	VAR jointtarget SDP_985 := [[-5.9, 34.76, 7.91, 0, 47.34, -89.94], [9E9, 9E9, 9E9, 9E9, 9E9, 9E9]];
	VAR jointtarget SDP_986 := [[-5.86, 34.75, 7.91, 0, 47.34, -91.23], [9E9, 9E9, 9E9, 9E9, 9E9, 9E9]];
	VAR jointtarget SDP_987 := [[-5.83, 34.75, 7.91, 0, 47.34, -92.52], [9E9, 9E9, 9E9, 9E9, 9E9, 9E9]];
	VAR jointtarget SDP_988 := [[-5.79, 34.75, 7.92, 0, 47.33, -93.81], [9E9, 9E9, 9E9, 9E9, 9E9, 9E9]];
	VAR jointtarget SDP_989 := [[-5.76, 34.75, 7.92, 0, 47.33, -95.1], [9E9, 9E9, 9E9, 9E9, 9E9, 9E9]];
	VAR jointtarget SDP_990 := [[-4.6, 34.64, 8.11, 0, 47.25, -94.6], [9E9, 9E9, 9E9, 9E9, 9E9, 9E9]];
	VAR jointtarget SDP_991 := [[-3.43, 34.55, 8.26, 0, 47.19, -93.43], [9E9, 9E9, 9E9, 9E9, 9E9, 9E9]];
	VAR jointtarget SDP_992 := [[-2.26, 34.49, 8.36, 0, 47.15, -92.26], [9E9, 9E9, 9E9, 9E9, 9E9, 9E9]];
	VAR jointtarget SDP_993 := [[-1.09, 34.45, 8.42, 0, 47.13, -91.09], [9E9, 9E9, 9E9, 9E9, 9E9, 9E9]];
	VAR jointtarget SDP_994 := [[0.09, 34.44, 8.44, 0, 47.12, -89.91], [9E9, 9E9, 9E9, 9E9, 9E9, 9E9]];
	VAR jointtarget SDP_995 := [[1.26, 34.46, 8.41, 0, 47.13, -88.74], [9E9, 9E9, 9E9, 9E9, 9E9, 9E9]];
	VAR jointtarget SDP_996 := [[2.43, 34.5, 8.35, 0, 47.16, -87.57], [9E9, 9E9, 9E9, 9E9, 9E9, 9E9]];
	VAR jointtarget SDP_997 := [[3.6, 34.56, 8.24, 0, 47.2, -86.4], [9E9, 9E9, 9E9, 9E9, 9E9, 9E9]];
	VAR jointtarget SDP_998 := [[4.77, 34.65, 8.08, 0, 47.27, -85.23], [9E9, 9E9, 9E9, 9E9, 9E9, 9E9]];
	VAR jointtarget SDP_999 := [[5.93, 34.77, 7.89, 0, 47.35, -84.07], [9E9, 9E9, 9E9, 9E9, 9E9, 9E9]];
	VAR jointtarget SDP_1000 := [[6.27, 34.83, 7.77, 0, 47.39, -79.23], [9E9, 9E9, 9E9, 9E9, 9E9, 9E9]];
	VAR jointtarget SDP_1001 := [[6.6, 34.96, 7.56, 0, 47.48, -69.9], [9E9, 9E9, 9E9, 9E9, 9E9, 9E9]];
	VAR jointtarget SDP_1002 := [[6.9, 35.14, 7.25, 0, 47.61, -60.6], [9E9, 9E9, 9E9, 9E9, 9E9, 9E9]];
	VAR jointtarget SDP_1003 := [[7.17, 35.37, 6.86, 0, 47.77, -51.33], [9E9, 9E9, 9E9, 9E9, 9E9, 9E9]];
	VAR jointtarget SDP_1004 := [[7.4, 35.64, 6.4, 0, 47.96, -42.1], [9E9, 9E9, 9E9, 9E9, 9E9, 9E9]];
	VAR jointtarget SDP_1005 := [[7.59, 35.95, 5.86, 0, 48.18, -32.91], [9E9, 9E9, 9E9, 9E9, 9E9, 9E9]];
	VAR jointtarget SDP_1006 := [[7.73, 36.29, 5.28, 0, 48.43, -23.77], [9E9, 9E9, 9E9, 9E9, 9E9, 9E9]];
	VAR jointtarget SDP_1007 := [[7.82, 36.65, 4.66, 0, 48.69, -14.68], [9E9, 9E9, 9E9, 9E9, 9E9, 9E9]];
	VAR jointtarget SDP_1008 := [[7.85, 37.02, 4.02, 0, 48.95, -5.65], [9E9, 9E9, 9E9, 9E9, 9E9, 9E9]];
	VAR jointtarget SDP_1009 := [[7.83, 37.4, 3.38, 0, 49.23, 3.33], [9E9, 9E9, 9E9, 9E9, 9E9, 9E9]];
	VAR jointtarget SDP_1010 := [[7.68, 38.65, 1.21, 0, 50.14, 7.68], [9E9, 9E9, 9E9, 9E9, 9E9, 9E9]];
	VAR jointtarget SDP_1011 := [[7.54, 39.92, -1.01, 0, 51.09, 7.54], [9E9, 9E9, 9E9, 9E9, 9E9, 9E9]];
	VAR jointtarget SDP_1012 := [[7.4, 41.21, -3.27, 0, 52.06, 7.4], [9E9, 9E9, 9E9, 9E9, 9E9, 9E9]];
	VAR jointtarget SDP_1013 := [[7.26, 42.52, -5.58, 0, 53.06, 7.26], [9E9, 9E9, 9E9, 9E9, 9E9, 9E9]];
	VAR jointtarget SDP_1014 := [[7.13, 43.85, -7.95, 0, 54.1, 7.13], [9E9, 9E9, 9E9, 9E9, 9E9, 9E9]];
	VAR jointtarget SDP_1015 := [[7.01, 45.21, -10.38, 0, 55.16, 7.01], [9E9, 9E9, 9E9, 9E9, 9E9, 9E9]];
	VAR jointtarget SDP_1016 := [[6.89, 46.6, -12.87, 0, 56.27, 6.89], [9E9, 9E9, 9E9, 9E9, 9E9, 9E9]];
	VAR jointtarget SDP_1017 := [[6.77, 48.03, -15.44, 0, 57.41, 6.77], [9E9, 9E9, 9E9, 9E9, 9E9, 9E9]];
	VAR jointtarget SDP_1018 := [[6.66, 49.49, -18.09, 0, 58.6, 6.66], [9E9, 9E9, 9E9, 9E9, 9E9, 9E9]];
	VAR jointtarget SDP_1019 := [[6.55, 51, -20.83, 0, 59.83, 6.55], [9E9, 9E9, 9E9, 9E9, 9E9, 9E9]];
	VAR jointtarget SDP_1020 := [[6.55, 51.04, -20.91, 0, 59.87, 5.89], [9E9, 9E9, 9E9, 9E9, 9E9, 9E9]];
	VAR jointtarget SDP_1021 := [[6.55, 51.09, -20.99, 0, 59.91, 4.56], [9E9, 9E9, 9E9, 9E9, 9E9, 9E9]];
	VAR jointtarget SDP_1022 := [[6.55, 51.13, -21.08, 0, 59.94, 3.24], [9E9, 9E9, 9E9, 9E9, 9E9, 9E9]];
	VAR jointtarget SDP_1023 := [[6.54, 51.18, -21.16, 0, 59.98, 1.91], [9E9, 9E9, 9E9, 9E9, 9E9, 9E9]];
	VAR jointtarget SDP_1024 := [[6.54, 51.22, -21.24, 0, 60.02, 0.59], [9E9, 9E9, 9E9, 9E9, 9E9, 9E9]];
	VAR jointtarget SDP_1025 := [[6.54, 51.27, -21.32, 0, 60.06, -0.74], [9E9, 9E9, 9E9, 9E9, 9E9, 9E9]];
	VAR jointtarget SDP_1026 := [[6.55, 51.32, -21.41, 0, 60.09, -2.06], [9E9, 9E9, 9E9, 9E9, 9E9, 9E9]];
	VAR jointtarget SDP_1027 := [[6.55, 51.36, -21.49, 0, 60.13, -3.38], [9E9, 9E9, 9E9, 9E9, 9E9, 9E9]];
	VAR jointtarget SDP_1028 := [[6.55, 51.41, -21.57, 0, 60.17, -4.7], [9E9, 9E9, 9E9, 9E9, 9E9, 9E9]];
	VAR jointtarget SDP_1029 := [[6.55, 51.45, -21.66, 0, 60.21, -6.03], [9E9, 9E9, 9E9, 9E9, 9E9, 9E9]];
	VAR jointtarget SDP_1030 := [[6.57, 51.63, -21.99, 0, 60.36, -6.68], [9E9, 9E9, 9E9, 9E9, 9E9, 9E9]];
	VAR jointtarget SDP_1031 := [[6.58, 51.82, -22.33, 0, 60.51, -6.66], [9E9, 9E9, 9E9, 9E9, 9E9, 9E9]];
	VAR jointtarget SDP_1032 := [[6.59, 52, -22.66, 0, 60.66, -6.65], [9E9, 9E9, 9E9, 9E9, 9E9, 9E9]];
	VAR jointtarget SDP_1033 := [[6.6, 52.19, -23, 0, 60.81, -6.64], [9E9, 9E9, 9E9, 9E9, 9E9, 9E9]];
	VAR jointtarget SDP_1034 := [[6.62, 52.37, -23.34, 0, 60.97, -6.62], [9E9, 9E9, 9E9, 9E9, 9E9, 9E9]];
	VAR jointtarget SDP_1035 := [[6.63, 52.56, -23.68, 0, 61.12, -6.61], [9E9, 9E9, 9E9, 9E9, 9E9, 9E9]];
	VAR jointtarget SDP_1036 := [[6.64, 52.75, -24.03, 0, 61.28, -6.6], [9E9, 9E9, 9E9, 9E9, 9E9, 9E9]];
	VAR jointtarget SDP_1037 := [[6.65, 52.94, -24.37, 0, 61.44, -6.59], [9E9, 9E9, 9E9, 9E9, 9E9, 9E9]];
	VAR jointtarget SDP_1038 := [[6.67, 53.13, -24.72, 0, 61.59, -6.57], [9E9, 9E9, 9E9, 9E9, 9E9, 9E9]];
	VAR jointtarget SDP_1039 := [[6.68, 53.32, -25.07, 0, 61.75, -6.56], [9E9, 9E9, 9E9, 9E9, 9E9, 9E9]];
	VAR jointtarget SDP_1040 := [[6.66, 53.69, -25.75, 0, 62.06, 3.75], [9E9, 9E9, 9E9, 9E9, 9E9, 9E9]];
	VAR jointtarget SDP_1041 := [[6.58, 54.03, -26.38, 0, 62.35, 24.31], [9E9, 9E9, 9E9, 9E9, 9E9, 9E9]];
	VAR jointtarget SDP_1042 := [[6.43, 54.3, -26.87, 0, 62.58, 44.81], [9E9, 9E9, 9E9, 9E9, 9E9, 9E9]];
	VAR jointtarget SDP_1043 := [[6.24, 54.46, -27.17, 0, 62.71, 65.27], [9E9, 9E9, 9E9, 9E9, 9E9, 9E9]];
	VAR jointtarget SDP_1044 := [[6.04, 54.49, -27.22, 0, 62.73, 85.71], [9E9, 9E9, 9E9, 9E9, 9E9, 9E9]];
	VAR jointtarget SDP_1045 := [[5.84, 54.38, -27.02, 0, 62.64, 106.16], [9E9, 9E9, 9E9, 9E9, 9E9, 9E9]];
	VAR jointtarget SDP_1046 := [[5.67, 54.15, -26.6, 0, 62.45, 126.64], [9E9, 9E9, 9E9, 9E9, 9E9, 9E9]];
	VAR jointtarget SDP_1047 := [[5.56, 53.83, -26.02, 0, 62.19, 147.18], [9E9, 9E9, 9E9, 9E9, 9E9, 9E9]];
	VAR jointtarget SDP_1048 := [[5.52, 53.47, -25.35, 0, 61.88, 167.78], [9E9, 9E9, 9E9, 9E9, 9E9, 9E9]];
	VAR jointtarget SDP_1049 := [[5.55, 53.1, -24.68, 0, 61.57, 188.46], [9E9, 9E9, 9E9, 9E9, 9E9, 9E9]];
	VAR jointtarget SDP_1050 := [[5.58, 52.92, -24.34, 0, 61.42, 198.82], [9E9, 9E9, 9E9, 9E9, 9E9, 9E9]];
	VAR jointtarget SDP_1051 := [[5.62, 52.74, -24.02, 0, 61.27, 198.86], [9E9, 9E9, 9E9, 9E9, 9E9, 9E9]];
	VAR jointtarget SDP_1052 := [[5.65, 52.56, -23.69, 0, 61.13, 198.89], [9E9, 9E9, 9E9, 9E9, 9E9, 9E9]];
	VAR jointtarget SDP_1053 := [[5.69, 52.39, -23.36, 0, 60.98, 198.93], [9E9, 9E9, 9E9, 9E9, 9E9, 9E9]];
	VAR jointtarget SDP_1054 := [[5.72, 52.21, -23.04, 0, 60.83, 198.96], [9E9, 9E9, 9E9, 9E9, 9E9, 9E9]];
	VAR jointtarget SDP_1055 := [[5.76, 52.03, -22.72, 0, 60.68, 199], [9E9, 9E9, 9E9, 9E9, 9E9, 9E9]];
	VAR jointtarget SDP_1056 := [[5.79, 51.86, -22.4, 0, 60.54, 199.03], [9E9, 9E9, 9E9, 9E9, 9E9, 9E9]];
	VAR jointtarget SDP_1057 := [[5.83, 51.68, -22.08, 0, 60.39, 199.07], [9E9, 9E9, 9E9, 9E9, 9E9, 9E9]];
	VAR jointtarget SDP_1058 := [[5.87, 51.51, -21.76, 0, 60.25, 199.11], [9E9, 9E9, 9E9, 9E9, 9E9, 9E9]];
	VAR jointtarget SDP_1059 := [[5.9, 51.33, -21.44, 0, 60.11, 199.14], [9E9, 9E9, 9E9, 9E9, 9E9, 9E9]];
	VAR jointtarget SDP_1060 := [[5.91, 51.29, -21.36, 0, 60.07, 198.49], [9E9, 9E9, 9E9, 9E9, 9E9, 9E9]];
	VAR jointtarget SDP_1061 := [[5.92, 51.25, -21.28, 0, 60.04, 197.17], [9E9, 9E9, 9E9, 9E9, 9E9, 9E9]];
	VAR jointtarget SDP_1062 := [[5.93, 51.2, -21.2, 0, 60, 195.86], [9E9, 9E9, 9E9, 9E9, 9E9, 9E9]];
	VAR jointtarget SDP_1063 := [[5.93, 51.16, -21.12, 0, 59.96, 194.54], [9E9, 9E9, 9E9, 9E9, 9E9, 9E9]];
	VAR jointtarget SDP_1064 := [[5.94, 51.11, -21.04, 0, 59.93, 193.22], [9E9, 9E9, 9E9, 9E9, 9E9, 9E9]];
	VAR jointtarget SDP_1065 := [[5.94, 51.07, -20.96, 0, 59.89, 191.9], [9E9, 9E9, 9E9, 9E9, 9E9, 9E9]];
	VAR jointtarget SDP_1066 := [[5.95, 51.03, -20.88, 0, 59.85, 190.58], [9E9, 9E9, 9E9, 9E9, 9E9, 9E9]];
	VAR jointtarget SDP_1067 := [[5.95, 50.98, -20.8, 0, 59.82, 189.26], [9E9, 9E9, 9E9, 9E9, 9E9, 9E9]];
	VAR jointtarget SDP_1068 := [[5.96, 50.94, -20.72, 0, 59.78, 187.94], [9E9, 9E9, 9E9, 9E9, 9E9, 9E9]];
	VAR jointtarget SDP_1069 := [[5.96, 50.89, -20.64, 0, 59.74, 186.62], [9E9, 9E9, 9E9, 9E9, 9E9, 9E9]];
	VAR jointtarget SDP_1070 := [[6.05, 49.48, -18.07, 0, 58.59, 186.05], [9E9, 9E9, 9E9, 9E9, 9E9, 9E9]];
	VAR jointtarget SDP_1071 := [[6.15, 48.11, -15.58, 0, 57.48, 186.15], [9E9, 9E9, 9E9, 9E9, 9E9, 9E9]];
	VAR jointtarget SDP_1072 := [[6.25, 46.77, -13.17, 0, 56.4, 186.25], [9E9, 9E9, 9E9, 9E9, 9E9, 9E9]];
	VAR jointtarget SDP_1073 := [[6.35, 45.46, -10.82, 0, 55.36, 186.35], [9E9, 9E9, 9E9, 9E9, 9E9, 9E9]];
	VAR jointtarget SDP_1074 := [[6.46, 44.18, -8.53, 0, 54.35, 186.46], [9E9, 9E9, 9E9, 9E9, 9E9, 9E9]];
	VAR jointtarget SDP_1075 := [[6.56, 42.92, -6.29, 0, 53.37, 186.56], [9E9, 9E9, 9E9, 9E9, 9E9, 9E9]];
	VAR jointtarget SDP_1076 := [[6.68, 41.68, -4.11, 0, 52.43, 186.68], [9E9, 9E9, 9E9, 9E9, 9E9, 9E9]];
	VAR jointtarget SDP_1077 := [[6.79, 40.47, -1.97, 0, 51.5, 186.79], [9E9, 9E9, 9E9, 9E9, 9E9, 9E9]];
	VAR jointtarget SDP_1078 := [[6.91, 39.27, 0.13, 0, 50.6, 186.91], [9E9, 9E9, 9E9, 9E9, 9E9, 9E9]];
	VAR jointtarget SDP_1079 := [[7.04, 38.08, 2.19, 0, 49.73, 187.04], [9E9, 9E9, 9E9, 9E9, 9E9, 9E9]];
	VAR jointtarget SDP_1080 := [[7.05, 37.71, 2.84, 0, 49.45, 182.55], [9E9, 9E9, 9E9, 9E9, 9E9, 9E9]];
	VAR jointtarget SDP_1081 := [[7.02, 37.33, 3.48, 0, 49.18, 173.52], [9E9, 9E9, 9E9, 9E9, 9E9, 9E9]];
	VAR jointtarget SDP_1082 := [[6.93, 36.97, 4.11, 0, 48.92, 164.43], [9E9, 9E9, 9E9, 9E9, 9E9, 9E9]];
	VAR jointtarget SDP_1083 := [[6.78, 36.63, 4.69, 0, 48.68, 155.28], [9E9, 9E9, 9E9, 9E9, 9E9, 9E9]];
	VAR jointtarget SDP_1084 := [[6.6, 36.33, 5.22, 0, 48.45, 146.1], [9E9, 9E9, 9E9, 9E9, 9E9, 9E9]];
	VAR jointtarget SDP_1085 := [[6.36, 36.05, 5.69, 0, 48.26, 136.86], [9E9, 9E9, 9E9, 9E9, 9E9, 9E9]];
	VAR jointtarget SDP_1086 := [[6.09, 35.83, 6.08, 0, 48.1, 127.59], [9E9, 9E9, 9E9, 9E9, 9E9, 9E9]];
	VAR jointtarget SDP_1087 := [[5.79, 35.65, 6.38, 0, 47.97, 118.29], [9E9, 9E9, 9E9, 9E9, 9E9, 9E9]];
	VAR jointtarget SDP_1088 := [[5.47, 35.53, 6.58, 0, 47.89, 108.97], [9E9, 9E9, 9E9, 9E9, 9E9, 9E9]];
	VAR jointtarget SDP_1089 := [[5.13, 35.47, 6.69, 0, 47.84, 99.63], [9E9, 9E9, 9E9, 9E9, 9E9, 9E9]];
	VAR jointtarget SDP_1090 := [[4.07, 35.38, 6.85, 0, 47.78, 94.07], [9E9, 9E9, 9E9, 9E9, 9E9, 9E9]];
	VAR jointtarget SDP_1091 := [[3.01, 35.31, 6.97, 0, 47.73, 93.01], [9E9, 9E9, 9E9, 9E9, 9E9, 9E9]];
	VAR jointtarget SDP_1092 := [[1.95, 35.26, 7.05, 0, 47.69, 91.95], [9E9, 9E9, 9E9, 9E9, 9E9, 9E9]];
	VAR jointtarget SDP_1093 := [[0.89, 35.23, 7.1, 0, 47.67, 90.89], [9E9, 9E9, 9E9, 9E9, 9E9, 9E9]];
	VAR jointtarget SDP_1094 := [[-0.18, 35.22, 7.11, 0, 47.67, 89.82], [9E9, 9E9, 9E9, 9E9, 9E9, 9E9]];
	VAR jointtarget SDP_1095 := [[-1.24, 35.24, 7.09, 0, 47.68, 88.76], [9E9, 9E9, 9E9, 9E9, 9E9, 9E9]];
	VAR jointtarget SDP_1096 := [[-2.31, 35.27, 7.03, 0, 47.7, 87.69], [9E9, 9E9, 9E9, 9E9, 9E9, 9E9]];
	VAR jointtarget SDP_1097 := [[-3.37, 35.33, 6.93, 0, 47.74, 86.63], [9E9, 9E9, 9E9, 9E9, 9E9, 9E9]];
	VAR jointtarget SDP_1098 := [[-4.43, 35.41, 6.8, 0, 47.8, 85.57], [9E9, 9E9, 9E9, 9E9, 9E9, 9E9]];
	VAR jointtarget SDP_1099 := [[-5.48, 35.5, 6.63, 0, 47.87, 84.52], [9E9, 9E9, 9E9, 9E9, 9E9, 9E9]];
	VAR jointtarget SDP_1100 := [[-5.59, 35.51, 6.62, 0, 47.87, 86.6], [9E9, 9E9, 9E9, 9E9, 9E9, 9E9]];
	VAR jointtarget SDP_1101 := [[-5.71, 35.51, 6.62, 0, 47.87, 90.88], [9E9, 9E9, 9E9, 9E9, 9E9, 9E9]];
	VAR jointtarget SDP_1102 := [[-5.82, 35.5, 6.64, 0, 47.86, 95.15], [9E9, 9E9, 9E9, 9E9, 9E9, 9E9]];
	VAR jointtarget SDP_1103 := [[-5.93, 35.48, 6.67, 0, 47.85, 99.43], [9E9, 9E9, 9E9, 9E9, 9E9, 9E9]];
	VAR jointtarget SDP_1104 := [[-6.04, 35.45, 6.72, 0, 47.83, 103.71], [9E9, 9E9, 9E9, 9E9, 9E9, 9E9]];
	VAR jointtarget SDP_1105 := [[-6.14, 35.41, 6.79, 0, 47.8, 107.99], [9E9, 9E9, 9E9, 9E9, 9E9, 9E9]];
	VAR jointtarget SDP_1106 := [[-6.25, 35.37, 6.86, 0, 47.77, 112.27], [9E9, 9E9, 9E9, 9E9, 9E9, 9E9]];
	VAR jointtarget SDP_1107 := [[-6.35, 35.31, 6.96, 0, 47.73, 116.56], [9E9, 9E9, 9E9, 9E9, 9E9, 9E9]];
	VAR jointtarget SDP_1108 := [[-6.44, 35.25, 7.06, 0, 47.69, 120.85], [9E9, 9E9, 9E9, 9E9, 9E9, 9E9]];
	VAR jointtarget SDP_1109 := [[-6.54, 35.18, 7.18, 0, 47.64, 125.15], [9E9, 9E9, 9E9, 9E9, 9E9, 9E9]];
	VAR jointtarget SDP_1110 := [[-6.59, 35.14, 7.25, 0, 47.61, 127.29], [9E9, 9E9, 9E9, 9E9, 9E9, 9E9]];
	VAR jointtarget SDP_1111 := [[-6.64, 35.09, 7.33, 0, 47.58, 127.23], [9E9, 9E9, 9E9, 9E9, 9E9, 9E9]];
	VAR jointtarget SDP_1112 := [[-6.7, 35.05, 7.4, 0, 47.55, 127.18], [9E9, 9E9, 9E9, 9E9, 9E9, 9E9]];
	VAR jointtarget SDP_1113 := [[-6.75, 35.01, 7.48, 0, 47.52, 127.12], [9E9, 9E9, 9E9, 9E9, 9E9, 9E9]];
	VAR jointtarget SDP_1114 := [[-6.81, 34.96, 7.55, 0, 47.48, 127.07], [9E9, 9E9, 9E9, 9E9, 9E9, 9E9]];
	VAR jointtarget SDP_1115 := [[-6.86, 34.92, 7.63, 0, 47.45, 127.01], [9E9, 9E9, 9E9, 9E9, 9E9, 9E9]];
	VAR jointtarget SDP_1116 := [[-6.92, 34.88, 7.7, 0, 47.42, 126.96], [9E9, 9E9, 9E9, 9E9, 9E9, 9E9]];
	VAR jointtarget SDP_1117 := [[-6.97, 34.83, 7.77, 0, 47.39, 126.91], [9E9, 9E9, 9E9, 9E9, 9E9, 9E9]];
	VAR jointtarget SDP_1118 := [[-7.03, 34.79, 7.85, 0, 47.36, 126.85], [9E9, 9E9, 9E9, 9E9, 9E9, 9E9]];
	VAR jointtarget SDP_1119 := [[-7.08, 34.75, 7.92, 0, 47.33, 126.8], [9E9, 9E9, 9E9, 9E9, 9E9, 9E9]];
	VAR jointtarget SDP_1120 := [[-7.39, 34.61, 8.16, 0, 47.24, 113.1], [9E9, 9E9, 9E9, 9E9, 9E9, 9E9]];
	VAR jointtarget SDP_1121 := [[-7.72, 34.63, 8.12, 0, 47.25, 85.99], [9E9, 9E9, 9E9, 9E9, 9E9, 9E9]];
	VAR jointtarget SDP_1122 := [[-8.01, 34.81, 7.81, 0, 47.38, 58.93], [9E9, 9E9, 9E9, 9E9, 9E9, 9E9]];
	VAR jointtarget SDP_1123 := [[-8.18, 35.11, 7.3, 0, 47.59, 31.98], [9E9, 9E9, 9E9, 9E9, 9E9, 9E9]];
	VAR jointtarget SDP_1124 := [[-8.21, 35.46, 6.71, 0, 47.84, 5.18], [9E9, 9E9, 9E9, 9E9, 9E9, 9E9]];
	VAR jointtarget SDP_1125 := [[-8.09, 35.79, 6.14, 0, 48.07, -21.48], [9E9, 9E9, 9E9, 9E9, 9E9, 9E9]];
	VAR jointtarget SDP_1126 := [[-7.85, 36.02, 5.74, 0, 48.24, -48.01], [9E9, 9E9, 9E9, 9E9, 9E9, 9E9]];
	VAR jointtarget SDP_1127 := [[-7.53, 36.12, 5.58, 0, 48.3, -74.47], [9E9, 9E9, 9E9, 9E9, 9E9, 9E9]];
	VAR jointtarget SDP_1128 := [[-7.21, 36.05, 5.7, 0, 48.26, -100.93], [9E9, 9E9, 9E9, 9E9, 9E9, 9E9]];
	VAR jointtarget SDP_1129 := [[-6.96, 35.83, 6.06, 0, 48.1, -127.44], [9E9, 9E9, 9E9, 9E9, 9E9, 9E9]];
	VAR jointtarget SDP_1130 := [[-6.9, 35.76, 6.19, 0, 48.05, -140.78], [9E9, 9E9, 9E9, 9E9, 9E9, 9E9]];
	VAR jointtarget SDP_1131 := [[-6.85, 35.69, 6.31, 0, 48, -140.72], [9E9, 9E9, 9E9, 9E9, 9E9, 9E9]];
	VAR jointtarget SDP_1132 := [[-6.79, 35.62, 6.43, 0, 47.95, -140.67], [9E9, 9E9, 9E9, 9E9, 9E9, 9E9]];
	VAR jointtarget SDP_1133 := [[-6.74, 35.55, 6.55, 0, 47.9, -140.62], [9E9, 9E9, 9E9, 9E9, 9E9, 9E9]];
	VAR jointtarget SDP_1134 := [[-6.68, 35.48, 6.67, 0, 47.85, -140.56], [9E9, 9E9, 9E9, 9E9, 9E9, 9E9]];
	VAR jointtarget SDP_1135 := [[-6.63, 35.41, 6.8, 0, 47.8, -140.51], [9E9, 9E9, 9E9, 9E9, 9E9, 9E9]];
	VAR jointtarget SDP_1136 := [[-6.58, 35.34, 6.92, 0, 47.75, -140.45], [9E9, 9E9, 9E9, 9E9, 9E9, 9E9]];
	VAR jointtarget SDP_1137 := [[-6.52, 35.26, 7.04, 0, 47.7, -140.4], [9E9, 9E9, 9E9, 9E9, 9E9, 9E9]];
	VAR jointtarget SDP_1138 := [[-6.47, 35.19, 7.16, 0, 47.65, -140.34], [9E9, 9E9, 9E9, 9E9, 9E9, 9E9]];
	VAR jointtarget SDP_1139 := [[-6.41, 35.12, 7.28, 0, 47.6, -140.29], [9E9, 9E9, 9E9, 9E9, 9E9, 9E9]];
	VAR jointtarget SDP_1140 := [[-6.38, 35.09, 7.33, 0, 47.58, -139.16], [9E9, 9E9, 9E9, 9E9, 9E9, 9E9]];
	VAR jointtarget SDP_1141 := [[-6.36, 35.06, 7.38, 0, 47.55, -136.92], [9E9, 9E9, 9E9, 9E9, 9E9, 9E9]];
	VAR jointtarget SDP_1142 := [[-6.33, 35.03, 7.43, 0, 47.53, -134.69], [9E9, 9E9, 9E9, 9E9, 9E9, 9E9]];
	VAR jointtarget SDP_1143 := [[-6.3, 35, 7.48, 0, 47.51, -132.45], [9E9, 9E9, 9E9, 9E9, 9E9, 9E9]];
	VAR jointtarget SDP_1144 := [[-6.27, 34.98, 7.53, 0, 47.5, -130.22], [9E9, 9E9, 9E9, 9E9, 9E9, 9E9]];
	VAR jointtarget SDP_1145 := [[-6.24, 34.95, 7.57, 0, 47.48, -127.98], [9E9, 9E9, 9E9, 9E9, 9E9, 9E9]];
	VAR jointtarget SDP_1146 := [[-6.21, 34.92, 7.61, 0, 47.46, -125.74], [9E9, 9E9, 9E9, 9E9, 9E9, 9E9]];
	VAR jointtarget SDP_1147 := [[-6.18, 34.9, 7.65, 0, 47.45, -123.5], [9E9, 9E9, 9E9, 9E9, 9E9, 9E9]];
	VAR jointtarget SDP_1148 := [[-6.14, 34.88, 7.69, 0, 47.43, -121.26], [9E9, 9E9, 9E9, 9E9, 9E9, 9E9]];
	VAR jointtarget SDP_1149 := [[-6.11, 34.86, 7.72, 0, 47.42, -119.01], [9E9, 9E9, 9E9, 9E9, 9E9, 9E9]];
	VAR jointtarget SDP_1150 := [[-6.09, 34.85, 7.74, 0, 47.42, -117.89], [9E9, 9E9, 9E9, 9E9, 9E9, 9E9]];
	VAR jointtarget SDP_1151 := [[-6.07, 34.84, 7.75, 0, 47.41, -117.87], [9E9, 9E9, 9E9, 9E9, 9E9, 9E9]];
	VAR jointtarget SDP_1152 := [[-6.05, 34.83, 7.77, 0, 47.4, -117.86], [9E9, 9E9, 9E9, 9E9, 9E9, 9E9]];
	VAR jointtarget SDP_1153 := [[-6.04, 34.81, 7.79, 0, 47.4, -117.84], [9E9, 9E9, 9E9, 9E9, 9E9, 9E9]];
	VAR jointtarget SDP_1154 := [[-6.02, 34.8, 7.8, 0, 47.39, -117.82], [9E9, 9E9, 9E9, 9E9, 9E9, 9E9]];
	VAR jointtarget SDP_1155 := [[-6, 34.79, 7.82, 0, 47.39, -117.8], [9E9, 9E9, 9E9, 9E9, 9E9, 9E9]];
	VAR jointtarget SDP_1156 := [[-5.98, 34.78, 7.84, 0, 47.38, -117.79], [9E9, 9E9, 9E9, 9E9, 9E9, 9E9]];
	VAR jointtarget SDP_1157 := [[-5.97, 34.77, 7.85, 0, 47.37, -117.77], [9E9, 9E9, 9E9, 9E9, 9E9, 9E9]];
	VAR jointtarget SDP_1158 := [[-5.95, 34.76, 7.87, 0, 47.37, -117.75], [9E9, 9E9, 9E9, 9E9, 9E9, 9E9]];
	VAR jointtarget SDP_1159 := [[-5.93, 34.75, 7.89, 0, 47.36, -117.73], [9E9, 9E9, 9E9, 9E9, 9E9, 9E9]];
	VAR jointtarget SDP_1160 := [[-4.75, 34.64, 8.08, 0, 47.28, -94.75], [9E9, 9E9, 9E9, 9E9, 9E9, 9E9]];
	VAR jointtarget SDP_1161 := [[-3.57, 34.55, 8.24, 0, 47.22, -93.57], [9E9, 9E9, 9E9, 9E9, 9E9, 9E9]];
	VAR jointtarget SDP_1162 := [[-2.38, 34.48, 8.35, 0, 47.17, -92.38], [9E9, 9E9, 9E9, 9E9, 9E9, 9E9]];
	VAR jointtarget SDP_1163 := [[-1.19, 34.44, 8.41, 0, 47.14, -91.19], [9E9, 9E9, 9E9, 9E9, 9E9, 9E9]];
	VAR jointtarget SDP_1164 := [[0, 34.43, 8.44, 0, 47.14, -90], [9E9, 9E9, 9E9, 9E9, 9E9, 9E9]];
	VAR jointtarget SDP_1165 := [[1.19, 34.44, 8.41, 0, 47.14, -88.81], [9E9, 9E9, 9E9, 9E9, 9E9, 9E9]];
	VAR jointtarget SDP_1166 := [[2.38, 34.48, 8.35, 0, 47.17, -87.62], [9E9, 9E9, 9E9, 9E9, 9E9, 9E9]];
	VAR jointtarget SDP_1167 := [[3.57, 34.55, 8.24, 0, 47.22, -86.43], [9E9, 9E9, 9E9, 9E9, 9E9, 9E9]];
	VAR jointtarget SDP_1168 := [[4.75, 34.64, 8.08, 0, 47.28, -85.25], [9E9, 9E9, 9E9, 9E9, 9E9, 9E9]];
	VAR jointtarget SDP_1169 := [[5.93, 34.75, 7.89, 0, 47.36, -84.07], [9E9, 9E9, 9E9, 9E9, 9E9, 9E9]];
	VAR jointtarget SDP_1170 := [[6.27, 34.82, 7.77, 0, 47.41, -79.23], [9E9, 9E9, 9E9, 9E9, 9E9, 9E9]];
	VAR jointtarget SDP_1171 := [[6.6, 34.94, 7.56, 0, 47.5, -69.9], [9E9, 9E9, 9E9, 9E9, 9E9, 9E9]];
	VAR jointtarget SDP_1172 := [[6.9, 35.12, 7.25, 0, 47.62, -60.6], [9E9, 9E9, 9E9, 9E9, 9E9, 9E9]];
	VAR jointtarget SDP_1173 := [[7.17, 35.35, 6.86, 0, 47.79, -51.33], [9E9, 9E9, 9E9, 9E9, 9E9, 9E9]];
	VAR jointtarget SDP_1174 := [[7.4, 35.63, 6.39, 0, 47.98, -42.1], [9E9, 9E9, 9E9, 9E9, 9E9, 9E9]];
	VAR jointtarget SDP_1175 := [[7.59, 35.94, 5.86, 0, 48.2, -32.91], [9E9, 9E9, 9E9, 9E9, 9E9, 9E9]];
	VAR jointtarget SDP_1176 := [[7.73, 36.28, 5.28, 0, 48.44, -23.77], [9E9, 9E9, 9E9, 9E9, 9E9, 9E9]];
	VAR jointtarget SDP_1177 := [[7.82, 36.64, 4.66, 0, 48.7, -14.68], [9E9, 9E9, 9E9, 9E9, 9E9, 9E9]];
	VAR jointtarget SDP_1178 := [[7.85, 37.01, 4.02, 0, 48.97, -5.65], [9E9, 9E9, 9E9, 9E9, 9E9, 9E9]];
	VAR jointtarget SDP_1179 := [[7.83, 37.38, 3.38, 0, 49.24, 3.33], [9E9, 9E9, 9E9, 9E9, 9E9, 9E9]];
	VAR jointtarget SDP_1180 := [[7.68, 38.61, 1.24, 0, 50.14, 7.68], [9E9, 9E9, 9E9, 9E9, 9E9, 9E9]];
	VAR jointtarget SDP_1181 := [[7.54, 39.86, -0.93, 0, 51.07, 7.54], [9E9, 9E9, 9E9, 9E9, 9E9, 9E9]];
	VAR jointtarget SDP_1182 := [[7.4, 41.12, -3.15, 0, 52.02, 7.4], [9E9, 9E9, 9E9, 9E9, 9E9, 9E9]];
	VAR jointtarget SDP_1183 := [[7.27, 42.41, -5.42, 0, 53.01, 7.27], [9E9, 9E9, 9E9, 9E9, 9E9, 9E9]];
	VAR jointtarget SDP_1184 := [[7.15, 43.72, -7.74, 0, 54.02, 7.15], [9E9, 9E9, 9E9, 9E9, 9E9, 9E9]];
	VAR jointtarget SDP_1185 := [[7.02, 45.05, -10.12, 0, 55.06, 7.02], [9E9, 9E9, 9E9, 9E9, 9E9, 9E9]];
	VAR jointtarget SDP_1186 := [[6.9, 46.42, -12.56, 0, 56.14, 6.9], [9E9, 9E9, 9E9, 9E9, 9E9, 9E9]];
	VAR jointtarget SDP_1187 := [[6.79, 47.81, -15.07, 0, 57.26, 6.79], [9E9, 9E9, 9E9, 9E9, 9E9, 9E9]];
	VAR jointtarget SDP_1188 := [[6.68, 49.24, -17.66, 0, 58.42, 6.68], [9E9, 9E9, 9E9, 9E9, 9E9, 9E9]];
	VAR jointtarget SDP_1189 := [[6.57, 50.72, -20.34, 0, 59.62, 6.57], [9E9, 9E9, 9E9, 9E9, 9E9, 9E9]];
	VAR jointtarget SDP_1190 := [[6.56, 50.86, -20.6, 0, 59.74, 8.75], [9E9, 9E9, 9E9, 9E9, 9E9, 9E9]];
	VAR jointtarget SDP_1191 := [[6.54, 51.01, -20.87, 0, 59.86, 13.12], [9E9, 9E9, 9E9, 9E9, 9E9, 9E9]];
	VAR jointtarget SDP_1192 := [[6.51, 51.15, -21.13, 0, 59.98, 17.48], [9E9, 9E9, 9E9, 9E9, 9E9, 9E9]];
	VAR jointtarget SDP_1193 := [[6.48, 51.29, -21.39, 0, 60.09, 21.83], [9E9, 9E9, 9E9, 9E9, 9E9, 9E9]];
	VAR jointtarget SDP_1194 := [[6.44, 51.43, -21.63, 0, 60.21, 26.18], [9E9, 9E9, 9E9, 9E9, 9E9, 9E9]];
	VAR jointtarget SDP_1195 := [[6.39, 51.56, -21.87, 0, 60.31, 30.52], [9E9, 9E9, 9E9, 9E9, 9E9, 9E9]];
	VAR jointtarget SDP_1196 := [[6.34, 51.68, -22.1, 0, 60.42, 34.86], [9E9, 9E9, 9E9, 9E9, 9E9, 9E9]];
	VAR jointtarget SDP_1197 := [[6.28, 51.8, -22.31, 0, 60.51, 39.19], [9E9, 9E9, 9E9, 9E9, 9E9, 9E9]];
	VAR jointtarget SDP_1198 := [[6.22, 51.91, -22.51, 0, 60.61, 43.51], [9E9, 9E9, 9E9, 9E9, 9E9, 9E9]];
	VAR jointtarget SDP_1199 := [[6.15, 52.01, -22.7, 0, 60.69, 47.83], [9E9, 9E9, 9E9, 9E9, 9E9, 9E9]];
	VAR jointtarget SDP_1200 := [[6.11, 52.07, -22.81, 0, 60.74, 49.99], [9E9, 9E9, 9E9, 9E9, 9E9, 9E9]];
	VAR jointtarget SDP_1201 := [[6.07, 52.13, -22.92, 0, 60.79, 49.95], [9E9, 9E9, 9E9, 9E9, 9E9, 9E9]];
	VAR jointtarget SDP_1202 := [[6.03, 52.19, -23.03, 0, 60.84, 49.9], [9E9, 9E9, 9E9, 9E9, 9E9, 9E9]];
	VAR jointtarget SDP_1203 := [[5.99, 52.25, -23.14, 0, 60.89, 49.86], [9E9, 9E9, 9E9, 9E9, 9E9, 9E9]];
	VAR jointtarget SDP_1204 := [[5.94, 52.31, -23.25, 0, 60.94, 49.82], [9E9, 9E9, 9E9, 9E9, 9E9, 9E9]];
	VAR jointtarget SDP_1205 := [[5.9, 52.37, -23.36, 0, 60.99, 49.78], [9E9, 9E9, 9E9, 9E9, 9E9, 9E9]];
	VAR jointtarget SDP_1206 := [[5.86, 52.43, -23.47, 0, 61.04, 49.74], [9E9, 9E9, 9E9, 9E9, 9E9, 9E9]];
	VAR jointtarget SDP_1207 := [[5.82, 52.49, -23.58, 0, 61.09, 49.7], [9E9, 9E9, 9E9, 9E9, 9E9, 9E9]];
	VAR jointtarget SDP_1208 := [[5.78, 52.55, -23.69, 0, 61.14, 49.66], [9E9, 9E9, 9E9, 9E9, 9E9, 9E9]];
	VAR jointtarget SDP_1209 := [[5.74, 52.61, -23.8, 0, 61.19, 49.61], [9E9, 9E9, 9E9, 9E9, 9E9, 9E9]];
	VAR jointtarget SDP_1210 := [[5.58, 52.98, -24.48, 0, 61.5, 36.07], [9E9, 9E9, 9E9, 9E9, 9E9, 9E9]];
	VAR jointtarget SDP_1211 := [[5.54, 53.44, -25.31, 0, 61.88, 9.25], [9E9, 9E9, 9E9, 9E9, 9E9, 9E9]];
	VAR jointtarget SDP_1212 := [[5.62, 53.88, -26.13, 0, 62.25, -17.44], [9E9, 9E9, 9E9, 9E9, 9E9, 9E9]];
	VAR jointtarget SDP_1213 := [[5.8, 54.22, -26.75, 0, 62.53, -44.04], [9E9, 9E9, 9E9, 9E9, 9E9, 9E9]];
	VAR jointtarget SDP_1214 := [[6.04, 54.38, -27.04, 0, 62.66, -70.57], [9E9, 9E9, 9E9, 9E9, 9E9, 9E9]];
	VAR jointtarget SDP_1215 := [[6.3, 54.32, -26.93, 0, 62.61, -97.09], [9E9, 9E9, 9E9, 9E9, 9E9, 9E9]];
	VAR jointtarget SDP_1216 := [[6.51, 54.06, -26.45, 0, 62.39, -123.65], [9E9, 9E9, 9E9, 9E9, 9E9, 9E9]];
	VAR jointtarget SDP_1217 := [[6.64, 53.65, -25.7, 0, 62.05, -150.3], [9E9, 9E9, 9E9, 9E9, 9E9, 9E9]];
	VAR jointtarget SDP_1218 := [[6.66, 53.18, -24.85, 0, 61.66, -177.06], [9E9, 9E9, 9E9, 9E9, 9E9, 9E9]];
	VAR jointtarget SDP_1219 := [[6.55, 52.76, -24.08, 0, 61.31, -203.94], [9E9, 9E9, 9E9, 9E9, 9E9, 9E9]];
	VAR jointtarget SDP_1220 := [[6.52, 52.69, -23.94, 0, 61.25, -217.36], [9E9, 9E9, 9E9, 9E9, 9E9, 9E9]];
	VAR jointtarget SDP_1221 := [[6.48, 52.62, -23.81, 0, 61.19, -217.39], [9E9, 9E9, 9E9, 9E9, 9E9, 9E9]];
	VAR jointtarget SDP_1222 := [[6.45, 52.54, -23.67, 0, 61.13, -217.42], [9E9, 9E9, 9E9, 9E9, 9E9, 9E9]];
	VAR jointtarget SDP_1223 := [[6.42, 52.47, -23.53, 0, 61.07, -217.46], [9E9, 9E9, 9E9, 9E9, 9E9, 9E9]];
	VAR jointtarget SDP_1224 := [[6.39, 52.39, -23.4, 0, 61.01, -217.49], [9E9, 9E9, 9E9, 9E9, 9E9, 9E9]];
	VAR jointtarget SDP_1225 := [[6.35, 52.32, -23.26, 0, 60.94, -217.52], [9E9, 9E9, 9E9, 9E9, 9E9, 9E9]];
	VAR jointtarget SDP_1226 := [[6.32, 52.24, -23.13, 0, 60.88, -217.56], [9E9, 9E9, 9E9, 9E9, 9E9, 9E9]];
	VAR jointtarget SDP_1227 := [[6.29, 52.17, -22.99, 0, 60.82, -217.59], [9E9, 9E9, 9E9, 9E9, 9E9, 9E9]];
	VAR jointtarget SDP_1228 := [[6.25, 52.1, -22.86, 0, 60.76, -217.62], [9E9, 9E9, 9E9, 9E9, 9E9, 9E9]];
	VAR jointtarget SDP_1229 := [[6.22, 52.02, -22.72, 0, 60.7, -217.66], [9E9, 9E9, 9E9, 9E9, 9E9, 9E9]];
	VAR jointtarget SDP_1230 := [[6.17, 51.9, -22.5, 0, 60.6, -215.51], [9E9, 9E9, 9E9, 9E9, 9E9, 9E9]];
	VAR jointtarget SDP_1231 := [[6.12, 51.77, -22.26, 0, 60.49, -211.17], [9E9, 9E9, 9E9, 9E9, 9E9, 9E9]];
	VAR jointtarget SDP_1232 := [[6.08, 51.63, -22.01, 0, 60.38, -206.83], [9E9, 9E9, 9E9, 9E9, 9E9, 9E9]];
	VAR jointtarget SDP_1233 := [[6.05, 51.49, -21.76, 0, 60.26, -202.47], [9E9, 9E9, 9E9, 9E9, 9E9, 9E9]];
	VAR jointtarget SDP_1234 := [[6.02, 51.35, -21.49, 0, 60.14, -198.11], [9E9, 9E9, 9E9, 9E9, 9E9, 9E9]];
	VAR jointtarget SDP_1235 := [[6, 51.2, -21.23, 0, 60.02, -193.75], [9E9, 9E9, 9E9, 9E9, 9E9, 9E9]];
	VAR jointtarget SDP_1236 := [[5.98, 51.06, -20.96, 0, 59.9, -189.38], [9E9, 9E9, 9E9, 9E9, 9E9, 9E9]];
	VAR jointtarget SDP_1237 := [[5.97, 50.91, -20.69, 0, 59.78, -185], [9E9, 9E9, 9E9, 9E9, 9E9, 9E9]];
	VAR jointtarget SDP_1238 := [[5.97, 50.76, -20.41, 0, 59.66, -180.61], [9E9, 9E9, 9E9, 9E9, 9E9, 9E9]];
	VAR jointtarget SDP_1239 := [[5.98, 50.61, -20.14, 0, 59.53, -176.22], [9E9, 9E9, 9E9, 9E9, 9E9, 9E9]];
	VAR jointtarget SDP_1240 := [[6.07, 49.23, -17.64, 0, 58.41, -173.93], [9E9, 9E9, 9E9, 9E9, 9E9, 9E9]];
	VAR jointtarget SDP_1241 := [[6.16, 47.89, -15.21, 0, 57.32, -173.84], [9E9, 9E9, 9E9, 9E9, 9E9, 9E9]];
	VAR jointtarget SDP_1242 := [[6.26, 46.58, -12.85, 0, 56.27, -173.74], [9E9, 9E9, 9E9, 9E9, 9E9, 9E9]];
	VAR jointtarget SDP_1243 := [[6.36, 45.3, -10.56, 0, 55.26, -173.64], [9E9, 9E9, 9E9, 9E9, 9E9, 9E9]];
	VAR jointtarget SDP_1244 := [[6.47, 44.04, -8.32, 0, 54.27, -173.53], [9E9, 9E9, 9E9, 9E9, 9E9, 9E9]];
	VAR jointtarget SDP_1245 := [[6.57, 42.81, -6.13, 0, 53.32, -173.43], [9E9, 9E9, 9E9, 9E9, 9E9, 9E9]];
	VAR jointtarget SDP_1246 := [[6.68, 41.6, -3.99, 0, 52.39, -173.32], [9E9, 9E9, 9E9, 9E9, 9E9, 9E9]];
	VAR jointtarget SDP_1247 := [[6.8, 40.41, -1.89, 0, 51.48, -173.2], [9E9, 9E9, 9E9, 9E9, 9E9, 9E9]];
	VAR jointtarget SDP_1248 := [[6.92, 39.23, 0.17, 0, 50.6, -173.08], [9E9, 9E9, 9E9, 9E9, 9E9, 9E9]];
	VAR jointtarget SDP_1249 := [[7.04, 38.07, 2.18, 0, 49.74, -172.96], [9E9, 9E9, 9E9, 9E9, 9E9, 9E9]];
	VAR jointtarget SDP_1250 := [[7.05, 37.7, 2.84, 0, 49.47, -177.45], [9E9, 9E9, 9E9, 9E9, 9E9, 9E9]];
	VAR jointtarget SDP_1251 := [[7.02, 37.32, 3.48, 0, 49.2, -186.48], [9E9, 9E9, 9E9, 9E9, 9E9, 9E9]];
	VAR jointtarget SDP_1252 := [[6.93, 36.96, 4.1, 0, 48.94, -195.57], [9E9, 9E9, 9E9, 9E9, 9E9, 9E9]];
	VAR jointtarget SDP_1253 := [[6.78, 36.62, 4.69, 0, 48.69, -204.72], [9E9, 9E9, 9E9, 9E9, 9E9, 9E9]];
	VAR jointtarget SDP_1254 := [[6.6, 36.31, 5.22, 0, 48.47, -213.9], [9E9, 9E9, 9E9, 9E9, 9E9, 9E9]];
	VAR jointtarget SDP_1255 := [[6.36, 36.04, 5.68, 0, 48.27, -223.14], [9E9, 9E9, 9E9, 9E9, 9E9, 9E9]];
	VAR jointtarget SDP_1256 := [[6.09, 35.81, 6.07, 0, 48.11, -232.41], [9E9, 9E9, 9E9, 9E9, 9E9, 9E9]];
	VAR jointtarget SDP_1257 := [[5.79, 35.64, 6.37, 0, 47.99, -241.71], [9E9, 9E9, 9E9, 9E9, 9E9, 9E9]];
	VAR jointtarget SDP_1258 := [[5.47, 35.52, 6.58, 0, 47.9, -251.03], [9E9, 9E9, 9E9, 9E9, 9E9, 9E9]];
	VAR jointtarget SDP_1259 := [[5.13, 35.45, 6.69, 0, 47.86, -260.37], [9E9, 9E9, 9E9, 9E9, 9E9, 9E9]];
	VAR jointtarget SDP_1260 := [[4.05, 35.36, 6.85, 0, 47.79, -265.95], [9E9, 9E9, 9E9, 9E9, 9E9, 9E9]];
	VAR jointtarget SDP_1261 := [[2.97, 35.29, 6.97, 0, 47.74, -267.03], [9E9, 9E9, 9E9, 9E9, 9E9, 9E9]];
	VAR jointtarget SDP_1262 := [[1.89, 35.24, 7.05, 0, 47.71, -268.11], [9E9, 9E9, 9E9, 9E9, 9E9, 9E9]];
	VAR jointtarget SDP_1263 := [[0.8, 35.22, 7.1, 0, 47.69, -269.2], [9E9, 9E9, 9E9, 9E9, 9E9, 9E9]];
	VAR jointtarget SDP_1264 := [[-0.28, 35.21, 7.11, 0, 47.68, -270.28], [9E9, 9E9, 9E9, 9E9, 9E9, 9E9]];
	VAR jointtarget SDP_1265 := [[-1.37, 35.23, 7.08, 0, 47.7, -271.37], [9E9, 9E9, 9E9, 9E9, 9E9, 9E9]];
	VAR jointtarget SDP_1266 := [[-2.45, 35.27, 7.01, 0, 47.72, -272.45], [9E9, 9E9, 9E9, 9E9, 9E9, 9E9]];
	VAR jointtarget SDP_1267 := [[-3.53, 35.33, 6.91, 0, 47.77, -273.53], [9E9, 9E9, 9E9, 9E9, 9E9, 9E9]];
	VAR jointtarget SDP_1268 := [[-4.61, 35.41, 6.77, 0, 47.82, -274.61], [9E9, 9E9, 9E9, 9E9, 9E9, 9E9]];
	VAR jointtarget SDP_1269 := [[-5.69, 35.51, 6.59, 0, 47.9, -275.69], [9E9, 9E9, 9E9, 9E9, 9E9, 9E9]];
	VAR jointtarget SDP_1270 := [[-5.72, 35.52, 6.58, 0, 47.9, -276.38], [9E9, 9E9, 9E9, 9E9, 9E9, 9E9]];
	VAR jointtarget SDP_1271 := [[-5.75, 35.52, 6.58, 0, 47.9, -277.74], [9E9, 9E9, 9E9, 9E9, 9E9, 9E9]];
	VAR jointtarget SDP_1272 := [[-5.79, 35.53, 6.57, 0, 47.91, -279.1], [9E9, 9E9, 9E9, 9E9, 9E9, 9E9]];
	VAR jointtarget SDP_1273 := [[-5.82, 35.53, 6.56, 0, 47.91, -280.46], [9E9, 9E9, 9E9, 9E9, 9E9, 9E9]];
	VAR jointtarget SDP_1274 := [[-5.85, 35.54, 6.54, 0, 47.92, -281.81], [9E9, 9E9, 9E9, 9E9, 9E9, 9E9]];
	VAR jointtarget SDP_1275 := [[-5.89, 35.55, 6.53, 0, 47.92, -283.17], [9E9, 9E9, 9E9, 9E9, 9E9, 9E9]];
	VAR jointtarget SDP_1276 := [[-5.92, 35.56, 6.51, 0, 47.93, -284.53], [9E9, 9E9, 9E9, 9E9, 9E9, 9E9]];
	VAR jointtarget SDP_1277 := [[-5.95, 35.57, 6.5, 0, 47.94, -285.88], [9E9, 9E9, 9E9, 9E9, 9E9, 9E9]];
	VAR jointtarget SDP_1278 := [[-5.98, 35.58, 6.48, 0, 47.94, -287.24], [9E9, 9E9, 9E9, 9E9, 9E9, 9E9]];
	VAR jointtarget SDP_1279 := [[-6.02, 35.59, 6.46, 0, 47.95, -288.59], [9E9, 9E9, 9E9, 9E9, 9E9, 9E9]];
	VAR jointtarget SDP_1280 := [[-6.14, 35.64, 6.38, 0, 47.99, -289.38], [9E9, 9E9, 9E9, 9E9, 9E9, 9E9]];
	VAR jointtarget SDP_1281 := [[-6.27, 35.69, 6.29, 0, 48.02, -289.51], [9E9, 9E9, 9E9, 9E9, 9E9, 9E9]];
	VAR jointtarget SDP_1282 := [[-6.4, 35.74, 6.21, 0, 48.06, -289.64], [9E9, 9E9, 9E9, 9E9, 9E9, 9E9]];
	VAR jointtarget SDP_1283 := [[-6.53, 35.79, 6.12, 0, 48.09, -289.77], [9E9, 9E9, 9E9, 9E9, 9E9, 9E9]];
	VAR jointtarget SDP_1284 := [[-6.66, 35.83, 6.04, 0, 48.13, -289.9], [9E9, 9E9, 9E9, 9E9, 9E9, 9E9]];
	VAR jointtarget SDP_1285 := [[-6.78, 35.88, 5.95, 0, 48.16, -290.02], [9E9, 9E9, 9E9, 9E9, 9E9, 9E9]];
	VAR jointtarget SDP_1286 := [[-6.91, 35.94, 5.87, 0, 48.2, -290.15], [9E9, 9E9, 9E9, 9E9, 9E9, 9E9]];
	VAR jointtarget SDP_1287 := [[-7.04, 35.99, 5.78, 0, 48.23, -290.28], [9E9, 9E9, 9E9, 9E9, 9E9, 9E9]];
	VAR jointtarget SDP_1288 := [[-7.16, 36.04, 5.69, 0, 48.27, -290.4], [9E9, 9E9, 9E9, 9E9, 9E9, 9E9]];
	VAR jointtarget SDP_1289 := [[-7.29, 36.09, 5.6, 0, 48.31, -290.53], [9E9, 9E9, 9E9, 9E9, 9E9, 9E9]];
	VAR jointtarget SDP_1290 := [[-7.55, 36.14, 5.52, 0, 48.34, -280.46], [9E9, 9E9, 9E9, 9E9, 9E9, 9E9]];
	VAR jointtarget SDP_1291 := [[-7.8, 36.09, 5.6, 0, 48.31, -260.07], [9E9, 9E9, 9E9, 9E9, 9E9, 9E9]];
	VAR jointtarget SDP_1292 := [[-8.03, 35.95, 5.85, 0, 48.21, -239.65], [9E9, 9E9, 9E9, 9E9, 9E9, 9E9]];
	VAR jointtarget SDP_1293 := [[-8.2, 35.73, 6.23, 0, 48.05, -219.17], [9E9, 9E9, 9E9, 9E9, 9E9, 9E9]];
	VAR jointtarget SDP_1294 := [[-8.28, 35.46, 6.68, 0, 47.86, -198.6], [9E9, 9E9, 9E9, 9E9, 9E9, 9E9]];
	VAR jointtarget SDP_1295 := [[-8.27, 35.17, 7.17, 0, 47.66, -177.95], [9E9, 9E9, 9E9, 9E9, 9E9, 9E9]];
	VAR jointtarget SDP_1296 := [[-8.17, 34.91, 7.61, 0, 47.48, -157.19], [9E9, 9E9, 9E9, 9E9, 9E9, 9E9]];
	VAR jointtarget SDP_1297 := [[-7.98, 34.71, 7.96, 0, 47.33, -136.36], [9E9, 9E9, 9E9, 9E9, 9E9, 9E9]];
	VAR jointtarget SDP_1298 := [[-7.74, 34.59, 8.16, 0, 47.25, -115.47], [9E9, 9E9, 9E9, 9E9, 9E9, 9E9]];
	VAR jointtarget SDP_1299 := [[-7.47, 34.57, 8.2, 0, 47.23, -94.56], [9E9, 9E9, 9E9, 9E9, 9E9, 9E9]];
	VAR jointtarget SDP_1300 := [[-7.34, 34.58, 8.18, 0, 47.24, -84.1], [9E9, 9E9, 9E9, 9E9, 9E9, 9E9]];
	VAR jointtarget SDP_1301 := [[-7.2, 34.59, 8.15, 0, 47.25, -83.96], [9E9, 9E9, 9E9, 9E9, 9E9, 9E9]];
	VAR jointtarget SDP_1302 := [[-7.06, 34.61, 8.13, 0, 47.27, -83.82], [9E9, 9E9, 9E9, 9E9, 9E9, 9E9]];
	VAR jointtarget SDP_1303 := [[-6.92, 34.62, 8.1, 0, 47.28, -83.68], [9E9, 9E9, 9E9, 9E9, 9E9, 9E9]];
	VAR jointtarget SDP_1304 := [[-6.79, 34.64, 8.07, 0, 47.29, -83.55], [9E9, 9E9, 9E9, 9E9, 9E9, 9E9]];
	VAR jointtarget SDP_1305 := [[-6.65, 34.65, 8.04, 0, 47.31, -83.41], [9E9, 9E9, 9E9, 9E9, 9E9, 9E9]];
	VAR jointtarget SDP_1306 := [[-6.51, 34.67, 8.01, 0, 47.32, -83.27], [9E9, 9E9, 9E9, 9E9, 9E9, 9E9]];
	VAR jointtarget SDP_1307 := [[-6.38, 34.68, 7.98, 0, 47.33, -83.14], [9E9, 9E9, 9E9, 9E9, 9E9, 9E9]];
	VAR jointtarget SDP_1308 := [[-6.24, 34.7, 7.95, 0, 47.35, -83], [9E9, 9E9, 9E9, 9E9, 9E9, 9E9]];
	VAR jointtarget SDP_1309 := [[-6.1, 34.72, 7.92, 0, 47.36, -82.86], [9E9, 9E9, 9E9, 9E9, 9E9, 9E9]];
	VAR jointtarget SDP_1310 := [[-6.07, 34.72, 7.92, 0, 47.36, -83.49], [9E9, 9E9, 9E9, 9E9, 9E9, 9E9]];
	VAR jointtarget SDP_1311 := [[-6.03, 34.72, 7.91, 0, 47.37, -84.78], [9E9, 9E9, 9E9, 9E9, 9E9, 9E9]];
	VAR jointtarget SDP_1312 := [[-6, 34.73, 7.91, 0, 47.37, -86.07], [9E9, 9E9, 9E9, 9E9, 9E9, 9E9]];
	VAR jointtarget SDP_1313 := [[-5.97, 34.73, 7.9, 0, 47.37, -87.36], [9E9, 9E9, 9E9, 9E9, 9E9, 9E9]];
	VAR jointtarget SDP_1314 := [[-5.93, 34.73, 7.9, 0, 47.37, -88.65], [9E9, 9E9, 9E9, 9E9, 9E9, 9E9]];
	VAR jointtarget SDP_1315 := [[-5.9, 34.73, 7.9, 0, 47.37, -89.94], [9E9, 9E9, 9E9, 9E9, 9E9, 9E9]];
	VAR jointtarget SDP_1316 := [[-5.86, 34.73, 7.9, 0, 47.37, -91.23], [9E9, 9E9, 9E9, 9E9, 9E9, 9E9]];
	VAR jointtarget SDP_1317 := [[-5.83, 34.73, 7.91, 0, 47.37, -92.52], [9E9, 9E9, 9E9, 9E9, 9E9, 9E9]];
	VAR jointtarget SDP_1318 := [[-5.79, 34.72, 7.91, 0, 47.37, -93.81], [9E9, 9E9, 9E9, 9E9, 9E9, 9E9]];
	VAR jointtarget SDP_1319 := [[-5.76, 34.72, 7.92, 0, 47.36, -95.1], [9E9, 9E9, 9E9, 9E9, 9E9, 9E9]];
	VAR jointtarget SDP_1320 := [[-4.6, 34.61, 8.1, 0, 47.29, -94.6], [9E9, 9E9, 9E9, 9E9, 9E9, 9E9]];
	VAR jointtarget SDP_1321 := [[-3.43, 34.52, 8.25, 0, 47.23, -93.43], [9E9, 9E9, 9E9, 9E9, 9E9, 9E9]];
	VAR jointtarget SDP_1322 := [[-2.26, 34.46, 8.35, 0, 47.18, -92.26], [9E9, 9E9, 9E9, 9E9, 9E9, 9E9]];
	VAR jointtarget SDP_1323 := [[-1.09, 34.43, 8.41, 0, 47.16, -91.09], [9E9, 9E9, 9E9, 9E9, 9E9, 9E9]];
	VAR jointtarget SDP_1324 := [[0.09, 34.42, 8.43, 0, 47.15, -89.91], [9E9, 9E9, 9E9, 9E9, 9E9, 9E9]];
	VAR jointtarget SDP_1325 := [[1.26, 34.43, 8.41, 0, 47.16, -88.74], [9E9, 9E9, 9E9, 9E9, 9E9, 9E9]];
	VAR jointtarget SDP_1326 := [[2.43, 34.47, 8.34, 0, 47.19, -87.57], [9E9, 9E9, 9E9, 9E9, 9E9, 9E9]];
	VAR jointtarget SDP_1327 := [[3.6, 34.53, 8.23, 0, 47.23, -86.4], [9E9, 9E9, 9E9, 9E9, 9E9, 9E9]];
	VAR jointtarget SDP_1328 := [[4.77, 34.62, 8.08, 0, 47.3, -85.23], [9E9, 9E9, 9E9, 9E9, 9E9, 9E9]];
	VAR jointtarget SDP_1329 := [[5.93, 34.74, 7.88, 0, 47.38, -84.07], [9E9, 9E9, 9E9, 9E9, 9E9, 9E9]];
	VAR jointtarget SDP_1330 := [[6.27, 34.81, 7.77, 0, 47.42, -79.23], [9E9, 9E9, 9E9, 9E9, 9E9, 9E9]];
	VAR jointtarget SDP_1331 := [[6.6, 34.93, 7.56, 0, 47.51, -69.9], [9E9, 9E9, 9E9, 9E9, 9E9, 9E9]];
	VAR jointtarget SDP_1332 := [[6.9, 35.11, 7.25, 0, 47.64, -60.6], [9E9, 9E9, 9E9, 9E9, 9E9, 9E9]];
	VAR jointtarget SDP_1333 := [[7.17, 35.34, 6.86, 0, 47.8, -51.33], [9E9, 9E9, 9E9, 9E9, 9E9, 9E9]];
	VAR jointtarget SDP_1334 := [[7.4, 35.61, 6.39, 0, 47.99, -42.1], [9E9, 9E9, 9E9, 9E9, 9E9, 9E9]];
	VAR jointtarget SDP_1335 := [[7.59, 35.92, 5.86, 0, 48.22, -32.91], [9E9, 9E9, 9E9, 9E9, 9E9, 9E9]];
	VAR jointtarget SDP_1336 := [[7.73, 36.26, 5.28, 0, 48.46, -23.77], [9E9, 9E9, 9E9, 9E9, 9E9, 9E9]];
	VAR jointtarget SDP_1337 := [[7.82, 36.62, 4.66, 0, 48.72, -14.68], [9E9, 9E9, 9E9, 9E9, 9E9, 9E9]];
	VAR jointtarget SDP_1338 := [[7.85, 37, 4.02, 0, 48.98, -5.65], [9E9, 9E9, 9E9, 9E9, 9E9, 9E9]];
	VAR jointtarget SDP_1339 := [[7.83, 37.37, 3.37, 0, 49.26, 3.33], [9E9, 9E9, 9E9, 9E9, 9E9, 9E9]];
	VAR jointtarget SDP_1340 := [[7.68, 38.62, 1.2, 0, 50.17, 7.68], [9E9, 9E9, 9E9, 9E9, 9E9, 9E9]];
	VAR jointtarget SDP_1341 := [[7.54, 39.89, -1.01, 0, 51.12, 7.54], [9E9, 9E9, 9E9, 9E9, 9E9, 9E9]];
	VAR jointtarget SDP_1342 := [[7.4, 41.18, -3.27, 0, 52.09, 7.4], [9E9, 9E9, 9E9, 9E9, 9E9, 9E9]];
	VAR jointtarget SDP_1343 := [[7.26, 42.49, -5.59, 0, 53.09, 7.26], [9E9, 9E9, 9E9, 9E9, 9E9, 9E9]];
	VAR jointtarget SDP_1344 := [[7.13, 43.83, -7.95, 0, 54.13, 7.13], [9E9, 9E9, 9E9, 9E9, 9E9, 9E9]];
	VAR jointtarget SDP_1345 := [[7.01, 45.19, -10.38, 0, 55.19, 7.01], [9E9, 9E9, 9E9, 9E9, 9E9, 9E9]];
	VAR jointtarget SDP_1346 := [[6.89, 46.58, -12.88, 0, 56.3, 6.89], [9E9, 9E9, 9E9, 9E9, 9E9, 9E9]];
	VAR jointtarget SDP_1347 := [[6.77, 48.01, -15.44, 0, 57.44, 6.77], [9E9, 9E9, 9E9, 9E9, 9E9, 9E9]];
	VAR jointtarget SDP_1348 := [[6.66, 49.47, -18.09, 0, 58.62, 6.66], [9E9, 9E9, 9E9, 9E9, 9E9, 9E9]];
	VAR jointtarget SDP_1349 := [[6.55, 50.98, -20.84, 0, 59.86, 6.55], [9E9, 9E9, 9E9, 9E9, 9E9, 9E9]];
	VAR jointtarget SDP_1350 := [[6.55, 51.02, -20.92, 0, 59.89, 5.89], [9E9, 9E9, 9E9, 9E9, 9E9, 9E9]];
	VAR jointtarget SDP_1351 := [[6.55, 51.07, -21, 0, 59.93, 4.56], [9E9, 9E9, 9E9, 9E9, 9E9, 9E9]];
	VAR jointtarget SDP_1352 := [[6.55, 51.11, -21.08, 0, 59.97, 3.24], [9E9, 9E9, 9E9, 9E9, 9E9, 9E9]];
	VAR jointtarget SDP_1353 := [[6.54, 51.16, -21.16, 0, 60.01, 1.91], [9E9, 9E9, 9E9, 9E9, 9E9, 9E9]];
	VAR jointtarget SDP_1354 := [[6.54, 51.2, -21.25, 0, 60.04, 0.59], [9E9, 9E9, 9E9, 9E9, 9E9, 9E9]];
	VAR jointtarget SDP_1355 := [[6.54, 51.25, -21.33, 0, 60.08, -0.74], [9E9, 9E9, 9E9, 9E9, 9E9, 9E9]];
	VAR jointtarget SDP_1356 := [[6.55, 51.29, -21.41, 0, 60.12, -2.06], [9E9, 9E9, 9E9, 9E9, 9E9, 9E9]];
	VAR jointtarget SDP_1357 := [[6.55, 51.34, -21.5, 0, 60.16, -3.38], [9E9, 9E9, 9E9, 9E9, 9E9, 9E9]];
	VAR jointtarget SDP_1358 := [[6.55, 51.38, -21.58, 0, 60.19, -4.7], [9E9, 9E9, 9E9, 9E9, 9E9, 9E9]];
	VAR jointtarget SDP_1359 := [[6.55, 51.43, -21.66, 0, 60.23, -6.03], [9E9, 9E9, 9E9, 9E9, 9E9, 9E9]];
	VAR jointtarget SDP_1360 := [[6.57, 51.61, -22, 0, 60.38, -6.68], [9E9, 9E9, 9E9, 9E9, 9E9, 9E9]];
	VAR jointtarget SDP_1361 := [[6.58, 51.8, -22.33, 0, 60.53, -6.66], [9E9, 9E9, 9E9, 9E9, 9E9, 9E9]];
	VAR jointtarget SDP_1362 := [[6.59, 51.98, -22.67, 0, 60.69, -6.65], [9E9, 9E9, 9E9, 9E9, 9E9, 9E9]];
	VAR jointtarget SDP_1363 := [[6.6, 52.17, -23.01, 0, 60.84, -6.64], [9E9, 9E9, 9E9, 9E9, 9E9, 9E9]];
	VAR jointtarget SDP_1364 := [[6.62, 52.35, -23.35, 0, 60.99, -6.62], [9E9, 9E9, 9E9, 9E9, 9E9, 9E9]];
	VAR jointtarget SDP_1365 := [[6.63, 52.54, -23.69, 0, 61.15, -6.61], [9E9, 9E9, 9E9, 9E9, 9E9, 9E9]];
	VAR jointtarget SDP_1366 := [[6.64, 52.73, -24.03, 0, 61.31, -6.6], [9E9, 9E9, 9E9, 9E9, 9E9, 9E9]];
	VAR jointtarget SDP_1367 := [[6.65, 52.92, -24.38, 0, 61.46, -6.59], [9E9, 9E9, 9E9, 9E9, 9E9, 9E9]];
	VAR jointtarget SDP_1368 := [[6.67, 53.11, -24.72, 0, 61.62, -6.57], [9E9, 9E9, 9E9, 9E9, 9E9, 9E9]];
	VAR jointtarget SDP_1369 := [[6.68, 53.3, -25.07, 0, 61.78, -6.56], [9E9, 9E9, 9E9, 9E9, 9E9, 9E9]];
	VAR jointtarget SDP_1370 := [[6.66, 53.67, -25.76, 0, 62.09, 3.75], [9E9, 9E9, 9E9, 9E9, 9E9, 9E9]];
	VAR jointtarget SDP_1371 := [[6.58, 54.01, -26.39, 0, 62.38, 24.31], [9E9, 9E9, 9E9, 9E9, 9E9, 9E9]];
	VAR jointtarget SDP_1372 := [[6.43, 54.28, -26.88, 0, 62.6, 44.81], [9E9, 9E9, 9E9, 9E9, 9E9, 9E9]];
	VAR jointtarget SDP_1373 := [[6.24, 54.44, -27.17, 0, 62.73, 65.27], [9E9, 9E9, 9E9, 9E9, 9E9, 9E9]];
	VAR jointtarget SDP_1374 := [[6.04, 54.47, -27.22, 0, 62.76, 85.71], [9E9, 9E9, 9E9, 9E9, 9E9, 9E9]];
	VAR jointtarget SDP_1375 := [[5.84, 54.36, -27.03, 0, 62.67, 106.16], [9E9, 9E9, 9E9, 9E9, 9E9, 9E9]];
	VAR jointtarget SDP_1376 := [[5.67, 54.13, -26.61, 0, 62.48, 126.64], [9E9, 9E9, 9E9, 9E9, 9E9, 9E9]];
	VAR jointtarget SDP_1377 := [[5.56, 53.81, -26.03, 0, 62.21, 147.18], [9E9, 9E9, 9E9, 9E9, 9E9, 9E9]];
	VAR jointtarget SDP_1378 := [[5.52, 53.45, -25.35, 0, 61.91, 167.78], [9E9, 9E9, 9E9, 9E9, 9E9, 9E9]];
	VAR jointtarget SDP_1379 := [[5.55, 53.08, -24.68, 0, 61.6, 188.46], [9E9, 9E9, 9E9, 9E9, 9E9, 9E9]];
	VAR jointtarget SDP_1380 := [[5.58, 52.9, -24.35, 0, 61.45, 198.82], [9E9, 9E9, 9E9, 9E9, 9E9, 9E9]];
	VAR jointtarget SDP_1381 := [[5.62, 52.72, -24.02, 0, 61.3, 198.86], [9E9, 9E9, 9E9, 9E9, 9E9, 9E9]];
	VAR jointtarget SDP_1382 := [[5.65, 52.54, -23.69, 0, 61.15, 198.89], [9E9, 9E9, 9E9, 9E9, 9E9, 9E9]];
	VAR jointtarget SDP_1383 := [[5.69, 52.36, -23.37, 0, 61, 198.93], [9E9, 9E9, 9E9, 9E9, 9E9, 9E9]];
	VAR jointtarget SDP_1384 := [[5.72, 52.19, -23.04, 0, 60.86, 198.96], [9E9, 9E9, 9E9, 9E9, 9E9, 9E9]];
	VAR jointtarget SDP_1385 := [[5.76, 52.01, -22.72, 0, 60.71, 199], [9E9, 9E9, 9E9, 9E9, 9E9, 9E9]];
	VAR jointtarget SDP_1386 := [[5.79, 51.84, -22.4, 0, 60.57, 199.03], [9E9, 9E9, 9E9, 9E9, 9E9, 9E9]];
	VAR jointtarget SDP_1387 := [[5.83, 51.66, -22.08, 0, 60.42, 199.07], [9E9, 9E9, 9E9, 9E9, 9E9, 9E9]];
	VAR jointtarget SDP_1388 := [[5.87, 51.49, -21.76, 0, 60.28, 199.11], [9E9, 9E9, 9E9, 9E9, 9E9, 9E9]];
	VAR jointtarget SDP_1389 := [[5.9, 51.31, -21.45, 0, 60.13, 199.14], [9E9, 9E9, 9E9, 9E9, 9E9, 9E9]];
	VAR jointtarget SDP_1390 := [[5.91, 51.27, -21.37, 0, 60.1, 198.49], [9E9, 9E9, 9E9, 9E9, 9E9, 9E9]];
	VAR jointtarget SDP_1391 := [[5.92, 51.23, -21.29, 0, 60.06, 197.17], [9E9, 9E9, 9E9, 9E9, 9E9, 9E9]];
	VAR jointtarget SDP_1392 := [[5.93, 51.18, -21.21, 0, 60.03, 195.86], [9E9, 9E9, 9E9, 9E9, 9E9, 9E9]];
	VAR jointtarget SDP_1393 := [[5.93, 51.14, -21.13, 0, 59.99, 194.54], [9E9, 9E9, 9E9, 9E9, 9E9, 9E9]];
	VAR jointtarget SDP_1394 := [[5.94, 51.09, -21.05, 0, 59.95, 193.22], [9E9, 9E9, 9E9, 9E9, 9E9, 9E9]];
	VAR jointtarget SDP_1395 := [[5.94, 51.05, -20.97, 0, 59.92, 191.9], [9E9, 9E9, 9E9, 9E9, 9E9, 9E9]];
	VAR jointtarget SDP_1396 := [[5.95, 51.01, -20.89, 0, 59.88, 190.58], [9E9, 9E9, 9E9, 9E9, 9E9, 9E9]];
	VAR jointtarget SDP_1397 := [[5.95, 50.96, -20.8, 0, 59.84, 189.26], [9E9, 9E9, 9E9, 9E9, 9E9, 9E9]];
	VAR jointtarget SDP_1398 := [[5.96, 50.92, -20.72, 0, 59.81, 187.94], [9E9, 9E9, 9E9, 9E9, 9E9, 9E9]];
	VAR jointtarget SDP_1399 := [[5.96, 50.87, -20.64, 0, 59.77, 186.62], [9E9, 9E9, 9E9, 9E9, 9E9, 9E9]];
	VAR jointtarget SDP_1400 := [[6.05, 49.46, -18.07, 0, 58.62, 186.05], [9E9, 9E9, 9E9, 9E9, 9E9, 9E9]];
	VAR jointtarget SDP_1401 := [[6.15, 48.09, -15.59, 0, 57.5, 186.15], [9E9, 9E9, 9E9, 9E9, 9E9, 9E9]];
	VAR jointtarget SDP_1402 := [[6.25, 46.75, -13.17, 0, 56.43, 186.25], [9E9, 9E9, 9E9, 9E9, 9E9, 9E9]];
	VAR jointtarget SDP_1403 := [[6.35, 45.44, -10.82, 0, 55.39, 186.35], [9E9, 9E9, 9E9, 9E9, 9E9, 9E9]];
	VAR jointtarget SDP_1404 := [[6.46, 44.15, -8.53, 0, 54.38, 186.46], [9E9, 9E9, 9E9, 9E9, 9E9, 9E9]];
	VAR jointtarget SDP_1405 := [[6.56, 42.9, -6.3, 0, 53.4, 186.56], [9E9, 9E9, 9E9, 9E9, 9E9, 9E9]];
	VAR jointtarget SDP_1406 := [[6.68, 41.66, -4.11, 0, 52.45, 186.68], [9E9, 9E9, 9E9, 9E9, 9E9, 9E9]];
	VAR jointtarget SDP_1407 := [[6.79, 40.44, -1.97, 0, 51.53, 186.79], [9E9, 9E9, 9E9, 9E9, 9E9, 9E9]];
	VAR jointtarget SDP_1408 := [[6.91, 39.24, 0.12, 0, 50.63, 186.91], [9E9, 9E9, 9E9, 9E9, 9E9, 9E9]];
	VAR jointtarget SDP_1409 := [[7.04, 38.06, 2.18, 0, 49.76, 187.04], [9E9, 9E9, 9E9, 9E9, 9E9, 9E9]];
	VAR jointtarget SDP_1410 := [[7.05, 37.68, 2.83, 0, 49.48, 182.55], [9E9, 9E9, 9E9, 9E9, 9E9, 9E9]];
	VAR jointtarget SDP_1411 := [[7.02, 37.31, 3.48, 0, 49.21, 173.52], [9E9, 9E9, 9E9, 9E9, 9E9, 9E9]];
	VAR jointtarget SDP_1412 := [[6.93, 36.95, 4.1, 0, 48.95, 164.43], [9E9, 9E9, 9E9, 9E9, 9E9, 9E9]];
	VAR jointtarget SDP_1413 := [[6.78, 36.61, 4.69, 0, 48.71, 155.28], [9E9, 9E9, 9E9, 9E9, 9E9, 9E9]];
	VAR jointtarget SDP_1414 := [[6.6, 36.3, 5.22, 0, 48.48, 146.1], [9E9, 9E9, 9E9, 9E9, 9E9, 9E9]];
	VAR jointtarget SDP_1415 := [[6.36, 36.03, 5.68, 0, 48.29, 136.86], [9E9, 9E9, 9E9, 9E9, 9E9, 9E9]];
	VAR jointtarget SDP_1416 := [[6.09, 35.8, 6.07, 0, 48.13, 127.59], [9E9, 9E9, 9E9, 9E9, 9E9, 9E9]];
	VAR jointtarget SDP_1417 := [[5.79, 35.63, 6.37, 0, 48, 118.29], [9E9, 9E9, 9E9, 9E9, 9E9, 9E9]];
	VAR jointtarget SDP_1418 := [[5.47, 35.5, 6.58, 0, 47.92, 108.97], [9E9, 9E9, 9E9, 9E9, 9E9, 9E9]];
	VAR jointtarget SDP_1419 := [[5.13, 35.44, 6.69, 0, 47.87, 99.63], [9E9, 9E9, 9E9, 9E9, 9E9, 9E9]];
	VAR jointtarget SDP_1420 := [[4.07, 35.35, 6.84, 0, 47.81, 94.07], [9E9, 9E9, 9E9, 9E9, 9E9, 9E9]];
	VAR jointtarget SDP_1421 := [[3.01, 35.28, 6.96, 0, 47.76, 93.01], [9E9, 9E9, 9E9, 9E9, 9E9, 9E9]];
	VAR jointtarget SDP_1422 := [[1.95, 35.23, 7.05, 0, 47.72, 91.95], [9E9, 9E9, 9E9, 9E9, 9E9, 9E9]];
	VAR jointtarget SDP_1423 := [[0.89, 35.2, 7.09, 0, 47.7, 90.89], [9E9, 9E9, 9E9, 9E9, 9E9, 9E9]];
	VAR jointtarget SDP_1424 := [[-0.18, 35.2, 7.1, 0, 47.7, 89.82], [9E9, 9E9, 9E9, 9E9, 9E9, 9E9]];
	VAR jointtarget SDP_1425 := [[-1.24, 35.21, 7.08, 0, 47.71, 88.76], [9E9, 9E9, 9E9, 9E9, 9E9, 9E9]];
	VAR jointtarget SDP_1426 := [[-2.31, 35.25, 7.02, 0, 47.73, 87.69], [9E9, 9E9, 9E9, 9E9, 9E9, 9E9]];
	VAR jointtarget SDP_1427 := [[-3.37, 35.3, 6.93, 0, 47.77, 86.63], [9E9, 9E9, 9E9, 9E9, 9E9, 9E9]];
	VAR jointtarget SDP_1428 := [[-4.43, 35.38, 6.79, 0, 47.83, 85.57], [9E9, 9E9, 9E9, 9E9, 9E9, 9E9]];
	VAR jointtarget SDP_1429 := [[-5.48, 35.48, 6.63, 0, 47.9, 84.52], [9E9, 9E9, 9E9, 9E9, 9E9, 9E9]];
	VAR jointtarget SDP_1430 := [[-5.59, 35.48, 6.61, 0, 47.9, 86.6], [9E9, 9E9, 9E9, 9E9, 9E9, 9E9]];
	VAR jointtarget SDP_1431 := [[-5.71, 35.48, 6.62, 0, 47.9, 90.88], [9E9, 9E9, 9E9, 9E9, 9E9, 9E9]];
	VAR jointtarget SDP_1432 := [[-5.82, 35.47, 6.64, 0, 47.89, 95.15], [9E9, 9E9, 9E9, 9E9, 9E9, 9E9]];
	VAR jointtarget SDP_1433 := [[-5.93, 35.45, 6.67, 0, 47.88, 99.43], [9E9, 9E9, 9E9, 9E9, 9E9, 9E9]];
	VAR jointtarget SDP_1434 := [[-6.04, 35.42, 6.72, 0, 47.86, 103.71], [9E9, 9E9, 9E9, 9E9, 9E9, 9E9]];
	VAR jointtarget SDP_1435 := [[-6.14, 35.39, 6.78, 0, 47.83, 107.99], [9E9, 9E9, 9E9, 9E9, 9E9, 9E9]];
	VAR jointtarget SDP_1436 := [[-6.25, 35.34, 6.86, 0, 47.8, 112.27], [9E9, 9E9, 9E9, 9E9, 9E9, 9E9]];
	VAR jointtarget SDP_1437 := [[-6.35, 35.29, 6.95, 0, 47.76, 116.56], [9E9, 9E9, 9E9, 9E9, 9E9, 9E9]];
	VAR jointtarget SDP_1438 := [[-6.44, 35.22, 7.06, 0, 47.72, 120.85], [9E9, 9E9, 9E9, 9E9, 9E9, 9E9]];
	VAR jointtarget SDP_1439 := [[-6.54, 35.16, 7.17, 0, 47.67, 125.15], [9E9, 9E9, 9E9, 9E9, 9E9, 9E9]];
	VAR jointtarget SDP_1440 := [[-6.59, 35.11, 7.25, 0, 47.64, 127.29], [9E9, 9E9, 9E9, 9E9, 9E9, 9E9]];
	VAR jointtarget SDP_1441 := [[-6.64, 35.07, 7.32, 0, 47.61, 127.23], [9E9, 9E9, 9E9, 9E9, 9E9, 9E9]];
	VAR jointtarget SDP_1442 := [[-6.7, 35.02, 7.4, 0, 47.58, 127.18], [9E9, 9E9, 9E9, 9E9, 9E9, 9E9]];
	VAR jointtarget SDP_1443 := [[-6.75, 34.98, 7.47, 0, 47.55, 127.12], [9E9, 9E9, 9E9, 9E9, 9E9, 9E9]];
	VAR jointtarget SDP_1444 := [[-6.81, 34.94, 7.55, 0, 47.52, 127.07], [9E9, 9E9, 9E9, 9E9, 9E9, 9E9]];
	VAR jointtarget SDP_1445 := [[-6.86, 34.89, 7.62, 0, 47.49, 127.01], [9E9, 9E9, 9E9, 9E9, 9E9, 9E9]];
	VAR jointtarget SDP_1446 := [[-6.92, 34.85, 7.7, 0, 47.46, 126.96], [9E9, 9E9, 9E9, 9E9, 9E9, 9E9]];
	VAR jointtarget SDP_1447 := [[-6.97, 34.81, 7.77, 0, 47.42, 126.91], [9E9, 9E9, 9E9, 9E9, 9E9, 9E9]];
	VAR jointtarget SDP_1448 := [[-7.03, 34.76, 7.84, 0, 47.39, 126.85], [9E9, 9E9, 9E9, 9E9, 9E9, 9E9]];
	VAR jointtarget SDP_1449 := [[-7.08, 34.72, 7.92, 0, 47.36, 126.8], [9E9, 9E9, 9E9, 9E9, 9E9, 9E9]];
	VAR jointtarget SDP_1450 := [[-7.39, 34.58, 8.15, 0, 47.27, 113.1], [9E9, 9E9, 9E9, 9E9, 9E9, 9E9]];
	VAR jointtarget SDP_1451 := [[-7.72, 34.6, 8.11, 0, 47.28, 85.99], [9E9, 9E9, 9E9, 9E9, 9E9, 9E9]];
	VAR jointtarget SDP_1452 := [[-8.01, 34.78, 7.81, 0, 47.41, 58.93], [9E9, 9E9, 9E9, 9E9, 9E9, 9E9]];
	VAR jointtarget SDP_1453 := [[-8.18, 35.08, 7.3, 0, 47.62, 31.98], [9E9, 9E9, 9E9, 9E9, 9E9, 9E9]];
	VAR jointtarget SDP_1454 := [[-8.21, 35.43, 6.7, 0, 47.87, 5.18], [9E9, 9E9, 9E9, 9E9, 9E9, 9E9]];
	VAR jointtarget SDP_1455 := [[-8.09, 35.76, 6.14, 0, 48.1, -21.48], [9E9, 9E9, 9E9, 9E9, 9E9, 9E9]];
	VAR jointtarget SDP_1456 := [[-7.85, 36, 5.73, 0, 48.27, -48.01], [9E9, 9E9, 9E9, 9E9, 9E9, 9E9]];
	VAR jointtarget SDP_1457 := [[-7.53, 36.09, 5.57, 0, 48.34, -74.47], [9E9, 9E9, 9E9, 9E9, 9E9, 9E9]];
	VAR jointtarget SDP_1458 := [[-7.21, 36.02, 5.69, 0, 48.29, -100.93], [9E9, 9E9, 9E9, 9E9, 9E9, 9E9]];
	VAR jointtarget SDP_1459 := [[-6.96, 35.81, 6.06, 0, 48.13, -127.44], [9E9, 9E9, 9E9, 9E9, 9E9, 9E9]];
	VAR jointtarget SDP_1460 := [[-6.9, 35.74, 6.18, 0, 48.08, -140.78], [9E9, 9E9, 9E9, 9E9, 9E9, 9E9]];
	VAR jointtarget SDP_1461 := [[-6.85, 35.66, 6.3, 0, 48.03, -140.72], [9E9, 9E9, 9E9, 9E9, 9E9, 9E9]];
	VAR jointtarget SDP_1462 := [[-6.79, 35.59, 6.43, 0, 47.98, -140.67], [9E9, 9E9, 9E9, 9E9, 9E9, 9E9]];
	VAR jointtarget SDP_1463 := [[-6.74, 35.52, 6.55, 0, 47.93, -140.62], [9E9, 9E9, 9E9, 9E9, 9E9, 9E9]];
	VAR jointtarget SDP_1464 := [[-6.68, 35.45, 6.67, 0, 47.88, -140.56], [9E9, 9E9, 9E9, 9E9, 9E9, 9E9]];
	VAR jointtarget SDP_1465 := [[-6.63, 35.38, 6.79, 0, 47.83, -140.51], [9E9, 9E9, 9E9, 9E9, 9E9, 9E9]];
	VAR jointtarget SDP_1466 := [[-6.58, 35.31, 6.91, 0, 47.78, -140.45], [9E9, 9E9, 9E9, 9E9, 9E9, 9E9]];
	VAR jointtarget SDP_1467 := [[-6.52, 35.24, 7.03, 0, 47.73, -140.4], [9E9, 9E9, 9E9, 9E9, 9E9, 9E9]];
	VAR jointtarget SDP_1468 := [[-6.47, 35.17, 7.15, 0, 47.68, -140.34], [9E9, 9E9, 9E9, 9E9, 9E9, 9E9]];
	VAR jointtarget SDP_1469 := [[-6.41, 35.1, 7.27, 0, 47.63, -140.29], [9E9, 9E9, 9E9, 9E9, 9E9, 9E9]];
	VAR jointtarget SDP_1470 := [[-6.38, 35.07, 7.33, 0, 47.61, -139.16], [9E9, 9E9, 9E9, 9E9, 9E9, 9E9]];
	VAR jointtarget SDP_1471 := [[-6.36, 35.03, 7.38, 0, 47.59, -136.92], [9E9, 9E9, 9E9, 9E9, 9E9, 9E9]];
	VAR jointtarget SDP_1472 := [[-6.33, 35.01, 7.43, 0, 47.57, -134.69], [9E9, 9E9, 9E9, 9E9, 9E9, 9E9]];
	VAR jointtarget SDP_1473 := [[-6.3, 34.98, 7.48, 0, 47.55, -132.45], [9E9, 9E9, 9E9, 9E9, 9E9, 9E9]];
	VAR jointtarget SDP_1474 := [[-6.27, 34.95, 7.52, 0, 47.53, -130.22], [9E9, 9E9, 9E9, 9E9, 9E9, 9E9]];
	VAR jointtarget SDP_1475 := [[-6.24, 34.92, 7.57, 0, 47.51, -127.98], [9E9, 9E9, 9E9, 9E9, 9E9, 9E9]];
	VAR jointtarget SDP_1476 := [[-6.21, 34.9, 7.61, 0, 47.5, -125.74], [9E9, 9E9, 9E9, 9E9, 9E9, 9E9]];
	VAR jointtarget SDP_1477 := [[-6.18, 34.87, 7.65, 0, 47.48, -123.5], [9E9, 9E9, 9E9, 9E9, 9E9, 9E9]];
	VAR jointtarget SDP_1478 := [[-6.14, 34.85, 7.68, 0, 47.47, -121.26], [9E9, 9E9, 9E9, 9E9, 9E9, 9E9]];
	VAR jointtarget SDP_1479 := [[-6.11, 34.83, 7.72, 0, 47.45, -119.01], [9E9, 9E9, 9E9, 9E9, 9E9, 9E9]];
	VAR jointtarget SDP_1480 := [[-6.09, 34.82, 7.73, 0, 47.45, -117.89], [9E9, 9E9, 9E9, 9E9, 9E9, 9E9]];
	VAR jointtarget SDP_1481 := [[-6.07, 34.81, 7.75, 0, 47.44, -117.87], [9E9, 9E9, 9E9, 9E9, 9E9, 9E9]];
	VAR jointtarget SDP_1482 := [[-6.05, 34.8, 7.77, 0, 47.44, -117.86], [9E9, 9E9, 9E9, 9E9, 9E9, 9E9]];
	VAR jointtarget SDP_1483 := [[-6.04, 34.79, 7.78, 0, 47.43, -117.84], [9E9, 9E9, 9E9, 9E9, 9E9, 9E9]];
	VAR jointtarget SDP_1484 := [[-6.02, 34.78, 7.8, 0, 47.42, -117.82], [9E9, 9E9, 9E9, 9E9, 9E9, 9E9]];
	VAR jointtarget SDP_1485 := [[-6, 34.77, 7.82, 0, 47.42, -117.8], [9E9, 9E9, 9E9, 9E9, 9E9, 9E9]];
	VAR jointtarget SDP_1486 := [[-5.98, 34.76, 7.83, 0, 47.41, -117.79], [9E9, 9E9, 9E9, 9E9, 9E9, 9E9]];
	VAR jointtarget SDP_1487 := [[-5.97, 34.75, 7.85, 0, 47.4, -117.77], [9E9, 9E9, 9E9, 9E9, 9E9, 9E9]];
	VAR jointtarget SDP_1488 := [[-5.95, 34.74, 7.87, 0, 47.4, -117.75], [9E9, 9E9, 9E9, 9E9, 9E9, 9E9]];
	VAR jointtarget SDP_1489 := [[-5.93, 34.73, 7.88, 0, 47.39, -117.73], [9E9, 9E9, 9E9, 9E9, 9E9, 9E9]];
	VAR jointtarget SDP_1490 := [[-4.75, 34.61, 8.08, 0, 47.31, -94.75], [9E9, 9E9, 9E9, 9E9, 9E9, 9E9]];
	VAR jointtarget SDP_1491 := [[-3.57, 34.52, 8.23, 0, 47.25, -93.57], [9E9, 9E9, 9E9, 9E9, 9E9, 9E9]];
	VAR jointtarget SDP_1492 := [[-2.38, 34.45, 8.34, 0, 47.2, -92.38], [9E9, 9E9, 9E9, 9E9, 9E9, 9E9]];
	VAR jointtarget SDP_1493 := [[-1.19, 34.42, 8.41, 0, 47.18, -91.19], [9E9, 9E9, 9E9, 9E9, 9E9, 9E9]];
	VAR jointtarget SDP_1494 := [[0, 34.4, 8.43, 0, 47.17, -90], [9E9, 9E9, 9E9, 9E9, 9E9, 9E9]];
	VAR jointtarget SDP_1495 := [[1.19, 34.42, 8.41, 0, 47.18, -88.81], [9E9, 9E9, 9E9, 9E9, 9E9, 9E9]];
	VAR jointtarget SDP_1496 := [[2.38, 34.45, 8.34, 0, 47.2, -87.62], [9E9, 9E9, 9E9, 9E9, 9E9, 9E9]];
	VAR jointtarget SDP_1497 := [[3.57, 34.52, 8.23, 0, 47.25, -86.43], [9E9, 9E9, 9E9, 9E9, 9E9, 9E9]];
	VAR jointtarget SDP_1498 := [[4.75, 34.61, 8.08, 0, 47.31, -85.25], [9E9, 9E9, 9E9, 9E9, 9E9, 9E9]];
	VAR jointtarget SDP_1499 := [[5.93, 34.73, 7.88, 0, 47.39, -84.07], [9E9, 9E9, 9E9, 9E9, 9E9, 9E9]];
	VAR jointtarget SDP_1500 := [[6.27, 34.79, 7.77, 0, 47.44, -79.23], [9E9, 9E9, 9E9, 9E9, 9E9, 9E9]];
	VAR jointtarget SDP_1501 := [[6.6, 34.92, 7.55, 0, 47.53, -69.9], [9E9, 9E9, 9E9, 9E9, 9E9, 9E9]];
	VAR jointtarget SDP_1502 := [[6.9, 35.1, 7.25, 0, 47.65, -60.6], [9E9, 9E9, 9E9, 9E9, 9E9, 9E9]];
	VAR jointtarget SDP_1503 := [[7.17, 35.33, 6.86, 0, 47.82, -51.33], [9E9, 9E9, 9E9, 9E9, 9E9, 9E9]];
	VAR jointtarget SDP_1504 := [[7.4, 35.6, 6.39, 0, 48.01, -42.1], [9E9, 9E9, 9E9, 9E9, 9E9, 9E9]];
	VAR jointtarget SDP_1505 := [[7.59, 35.91, 5.86, 0, 48.23, -32.91], [9E9, 9E9, 9E9, 9E9, 9E9, 9E9]];
	VAR jointtarget SDP_1506 := [[7.73, 36.25, 5.28, 0, 48.47, -23.77], [9E9, 9E9, 9E9, 9E9, 9E9, 9E9]];
	VAR jointtarget SDP_1507 := [[7.82, 36.61, 4.66, 0, 48.73, -14.68], [9E9, 9E9, 9E9, 9E9, 9E9, 9E9]];
	VAR jointtarget SDP_1508 := [[7.85, 36.98, 4.02, 0, 49, -5.65], [9E9, 9E9, 9E9, 9E9, 9E9, 9E9]];
	VAR jointtarget SDP_1509 := [[7.83, 37.36, 3.37, 0, 49.27, 3.33], [9E9, 9E9, 9E9, 9E9, 9E9, 9E9]];
	VAR jointtarget SDP_1510 := [[7.68, 38.59, 1.24, 0, 50.17, 7.68], [9E9, 9E9, 9E9, 9E9, 9E9, 9E9]];
	VAR jointtarget SDP_1511 := [[7.54, 39.83, -0.93, 0, 51.1, 7.54], [9E9, 9E9, 9E9, 9E9, 9E9, 9E9]];
	VAR jointtarget SDP_1512 := [[7.4, 41.1, -3.15, 0, 52.05, 7.4], [9E9, 9E9, 9E9, 9E9, 9E9, 9E9]];
	VAR jointtarget SDP_1513 := [[7.27, 42.39, -5.42, 0, 53.03, 7.27], [9E9, 9E9, 9E9, 9E9, 9E9, 9E9]];
	VAR jointtarget SDP_1514 := [[7.15, 43.7, -7.74, 0, 54.05, 7.15], [9E9, 9E9, 9E9, 9E9, 9E9, 9E9]];
	VAR jointtarget SDP_1515 := [[7.02, 45.03, -10.12, 0, 55.09, 7.02], [9E9, 9E9, 9E9, 9E9, 9E9, 9E9]];
	VAR jointtarget SDP_1516 := [[6.9, 46.39, -12.56, 0, 56.17, 6.9], [9E9, 9E9, 9E9, 9E9, 9E9, 9E9]];
	VAR jointtarget SDP_1517 := [[6.79, 47.79, -15.08, 0, 57.29, 6.79], [9E9, 9E9, 9E9, 9E9, 9E9, 9E9]];
	VAR jointtarget SDP_1518 := [[6.68, 49.22, -17.67, 0, 58.44, 6.68], [9E9, 9E9, 9E9, 9E9, 9E9, 9E9]];
	VAR jointtarget SDP_1519 := [[6.57, 50.69, -20.34, 0, 59.65, 6.57], [9E9, 9E9, 9E9, 9E9, 9E9, 9E9]];
	VAR jointtarget SDP_1520 := [[6.56, 50.84, -20.61, 0, 59.77, 8.75], [9E9, 9E9, 9E9, 9E9, 9E9, 9E9]];
	VAR jointtarget SDP_1521 := [[6.54, 50.99, -20.88, 0, 59.89, 13.12], [9E9, 9E9, 9E9, 9E9, 9E9, 9E9]];
	VAR jointtarget SDP_1522 := [[6.51, 51.13, -21.14, 0, 60.01, 17.48], [9E9, 9E9, 9E9, 9E9, 9E9, 9E9]];
	VAR jointtarget SDP_1523 := [[6.48, 51.27, -21.39, 0, 60.12, 21.83], [9E9, 9E9, 9E9, 9E9, 9E9, 9E9]];
	VAR jointtarget SDP_1524 := [[6.44, 51.41, -21.64, 0, 60.23, 26.18], [9E9, 9E9, 9E9, 9E9, 9E9, 9E9]];
	VAR jointtarget SDP_1525 := [[6.39, 51.54, -21.88, 0, 60.34, 30.52], [9E9, 9E9, 9E9, 9E9, 9E9, 9E9]];
	VAR jointtarget SDP_1526 := [[6.34, 51.66, -22.1, 0, 60.44, 34.86], [9E9, 9E9, 9E9, 9E9, 9E9, 9E9]];
	VAR jointtarget SDP_1527 := [[6.28, 51.78, -22.32, 0, 60.54, 39.19], [9E9, 9E9, 9E9, 9E9, 9E9, 9E9]];
	VAR jointtarget SDP_1528 := [[6.22, 51.89, -22.52, 0, 60.63, 43.51], [9E9, 9E9, 9E9, 9E9, 9E9, 9E9]];
	VAR jointtarget SDP_1529 := [[6.15, 51.99, -22.71, 0, 60.72, 47.83], [9E9, 9E9, 9E9, 9E9, 9E9, 9E9]];
	VAR jointtarget SDP_1530 := [[6.11, 52.05, -22.82, 0, 60.77, 49.99], [9E9, 9E9, 9E9, 9E9, 9E9, 9E9]];
	VAR jointtarget SDP_1531 := [[6.07, 52.11, -22.92, 0, 60.81, 49.95], [9E9, 9E9, 9E9, 9E9, 9E9, 9E9]];
	VAR jointtarget SDP_1532 := [[6.03, 52.17, -23.03, 0, 60.86, 49.9], [9E9, 9E9, 9E9, 9E9, 9E9, 9E9]];
	VAR jointtarget SDP_1533 := [[5.99, 52.23, -23.14, 0, 60.91, 49.86], [9E9, 9E9, 9E9, 9E9, 9E9, 9E9]];
	VAR jointtarget SDP_1534 := [[5.94, 52.29, -23.25, 0, 60.96, 49.82], [9E9, 9E9, 9E9, 9E9, 9E9, 9E9]];
	VAR jointtarget SDP_1535 := [[5.9, 52.35, -23.36, 0, 61.01, 49.78], [9E9, 9E9, 9E9, 9E9, 9E9, 9E9]];
	VAR jointtarget SDP_1536 := [[5.86, 52.41, -23.47, 0, 61.06, 49.74], [9E9, 9E9, 9E9, 9E9, 9E9, 9E9]];
	VAR jointtarget SDP_1537 := [[5.82, 52.47, -23.58, 0, 61.11, 49.7], [9E9, 9E9, 9E9, 9E9, 9E9, 9E9]];
	VAR jointtarget SDP_1538 := [[5.78, 52.53, -23.7, 0, 61.16, 49.66], [9E9, 9E9, 9E9, 9E9, 9E9, 9E9]];
	VAR jointtarget SDP_1539 := [[5.74, 52.59, -23.81, 0, 61.21, 49.61], [9E9, 9E9, 9E9, 9E9, 9E9, 9E9]];
	VAR jointtarget SDP_1540 := [[5.58, 52.96, -24.48, 0, 61.52, 36.07], [9E9, 9E9, 9E9, 9E9, 9E9, 9E9]];
	VAR jointtarget SDP_1541 := [[5.54, 53.42, -25.32, 0, 61.9, 9.25], [9E9, 9E9, 9E9, 9E9, 9E9, 9E9]];
	VAR jointtarget SDP_1542 := [[5.62, 53.86, -26.14, 0, 62.27, -17.44], [9E9, 9E9, 9E9, 9E9, 9E9, 9E9]];
	VAR jointtarget SDP_1543 := [[5.8, 54.2, -26.76, 0, 62.56, -44.04], [9E9, 9E9, 9E9, 9E9, 9E9, 9E9]];
	VAR jointtarget SDP_1544 := [[6.04, 54.36, -27.05, 0, 62.69, -70.57], [9E9, 9E9, 9E9, 9E9, 9E9, 9E9]];
	VAR jointtarget SDP_1545 := [[6.3, 54.3, -26.94, 0, 62.64, -97.09], [9E9, 9E9, 9E9, 9E9, 9E9, 9E9]];
	VAR jointtarget SDP_1546 := [[6.51, 54.03, -26.45, 0, 62.42, -123.65], [9E9, 9E9, 9E9, 9E9, 9E9, 9E9]];
	VAR jointtarget SDP_1547 := [[6.64, 53.63, -25.7, 0, 62.08, -150.3], [9E9, 9E9, 9E9, 9E9, 9E9, 9E9]];
	VAR jointtarget SDP_1548 := [[6.66, 53.16, -24.85, 0, 61.69, -177.06], [9E9, 9E9, 9E9, 9E9, 9E9, 9E9]];
	VAR jointtarget SDP_1549 := [[6.55, 52.74, -24.08, 0, 61.34, -203.94], [9E9, 9E9, 9E9, 9E9, 9E9, 9E9]];
	VAR jointtarget SDP_1550 := [[6.52, 52.67, -23.95, 0, 61.28, -217.36], [9E9, 9E9, 9E9, 9E9, 9E9, 9E9]];
	VAR jointtarget SDP_1551 := [[6.48, 52.59, -23.81, 0, 61.22, -217.39], [9E9, 9E9, 9E9, 9E9, 9E9, 9E9]];
	VAR jointtarget SDP_1552 := [[6.45, 52.52, -23.67, 0, 61.15, -217.42], [9E9, 9E9, 9E9, 9E9, 9E9, 9E9]];
	VAR jointtarget SDP_1553 := [[6.42, 52.45, -23.54, 0, 61.09, -217.46], [9E9, 9E9, 9E9, 9E9, 9E9, 9E9]];
	VAR jointtarget SDP_1554 := [[6.39, 52.37, -23.4, 0, 61.03, -217.49], [9E9, 9E9, 9E9, 9E9, 9E9, 9E9]];
	VAR jointtarget SDP_1555 := [[6.35, 52.3, -23.27, 0, 60.97, -217.52], [9E9, 9E9, 9E9, 9E9, 9E9, 9E9]];
	VAR jointtarget SDP_1556 := [[6.32, 52.22, -23.13, 0, 60.91, -217.56], [9E9, 9E9, 9E9, 9E9, 9E9, 9E9]];
	VAR jointtarget SDP_1557 := [[6.29, 52.15, -23, 0, 60.85, -217.59], [9E9, 9E9, 9E9, 9E9, 9E9, 9E9]];
	VAR jointtarget SDP_1558 := [[6.25, 52.08, -22.86, 0, 60.79, -217.62], [9E9, 9E9, 9E9, 9E9, 9E9, 9E9]];
	VAR jointtarget SDP_1559 := [[6.22, 52, -22.73, 0, 60.73, -217.66], [9E9, 9E9, 9E9, 9E9, 9E9, 9E9]];
	VAR jointtarget SDP_1560 := [[6.17, 51.88, -22.5, 0, 60.62, -215.51], [9E9, 9E9, 9E9, 9E9, 9E9, 9E9]];
	VAR jointtarget SDP_1561 := [[6.12, 51.75, -22.26, 0, 60.52, -211.17], [9E9, 9E9, 9E9, 9E9, 9E9, 9E9]];
	VAR jointtarget SDP_1562 := [[6.08, 51.61, -22.02, 0, 60.4, -206.83], [9E9, 9E9, 9E9, 9E9, 9E9, 9E9]];
	VAR jointtarget SDP_1563 := [[6.05, 51.47, -21.76, 0, 60.29, -202.47], [9E9, 9E9, 9E9, 9E9, 9E9, 9E9]];
	VAR jointtarget SDP_1564 := [[6.02, 51.33, -21.5, 0, 60.17, -198.11], [9E9, 9E9, 9E9, 9E9, 9E9, 9E9]];
	VAR jointtarget SDP_1565 := [[6, 51.18, -21.23, 0, 60.05, -193.75], [9E9, 9E9, 9E9, 9E9, 9E9, 9E9]];
	VAR jointtarget SDP_1566 := [[5.98, 51.03, -20.96, 0, 59.93, -189.38], [9E9, 9E9, 9E9, 9E9, 9E9, 9E9]];
	VAR jointtarget SDP_1567 := [[5.97, 50.89, -20.69, 0, 59.8, -185], [9E9, 9E9, 9E9, 9E9, 9E9, 9E9]];
	VAR jointtarget SDP_1568 := [[5.97, 50.74, -20.42, 0, 59.68, -180.61], [9E9, 9E9, 9E9, 9E9, 9E9, 9E9]];
	VAR jointtarget SDP_1569 := [[5.98, 50.59, -20.15, 0, 59.56, -176.22], [9E9, 9E9, 9E9, 9E9, 9E9, 9E9]];
	VAR jointtarget SDP_1570 := [[6.07, 49.21, -17.65, 0, 58.43, -173.93], [9E9, 9E9, 9E9, 9E9, 9E9, 9E9]];
	VAR jointtarget SDP_1571 := [[6.16, 47.87, -15.22, 0, 57.35, -173.84], [9E9, 9E9, 9E9, 9E9, 9E9, 9E9]];
	VAR jointtarget SDP_1572 := [[6.26, 46.56, -12.86, 0, 56.3, -173.74], [9E9, 9E9, 9E9, 9E9, 9E9, 9E9]];
	VAR jointtarget SDP_1573 := [[6.36, 45.28, -10.56, 0, 55.28, -173.64], [9E9, 9E9, 9E9, 9E9, 9E9, 9E9]];
	VAR jointtarget SDP_1574 := [[6.47, 44.02, -8.32, 0, 54.3, -173.53], [9E9, 9E9, 9E9, 9E9, 9E9, 9E9]];
	VAR jointtarget SDP_1575 := [[6.57, 42.79, -6.13, 0, 53.34, -173.43], [9E9, 9E9, 9E9, 9E9, 9E9, 9E9]];
	VAR jointtarget SDP_1576 := [[6.68, 41.58, -3.99, 0, 52.41, -173.32], [9E9, 9E9, 9E9, 9E9, 9E9, 9E9]];
	VAR jointtarget SDP_1577 := [[6.8, 40.38, -1.89, 0, 51.51, -173.2], [9E9, 9E9, 9E9, 9E9, 9E9, 9E9]];
	VAR jointtarget SDP_1578 := [[6.92, 39.21, 0.16, 0, 50.63, -173.08], [9E9, 9E9, 9E9, 9E9, 9E9, 9E9]];
	VAR jointtarget SDP_1579 := [[7.04, 38.05, 2.18, 0, 49.77, -172.96], [9E9, 9E9, 9E9, 9E9, 9E9, 9E9]];
	VAR jointtarget SDP_1580 := [[7.05, 37.67, 2.83, 0, 49.5, -177.45], [9E9, 9E9, 9E9, 9E9, 9E9, 9E9]];
	VAR jointtarget SDP_1581 := [[7.02, 37.3, 3.48, 0, 49.23, -186.48], [9E9, 9E9, 9E9, 9E9, 9E9, 9E9]];
	VAR jointtarget SDP_1582 := [[6.93, 36.94, 4.1, 0, 48.97, -195.57], [9E9, 9E9, 9E9, 9E9, 9E9, 9E9]];
	VAR jointtarget SDP_1583 := [[6.78, 36.6, 4.68, 0, 48.72, -204.72], [9E9, 9E9, 9E9, 9E9, 9E9, 9E9]];
	VAR jointtarget SDP_1584 := [[6.6, 36.29, 5.21, 0, 48.5, -213.9], [9E9, 9E9, 9E9, 9E9, 9E9, 9E9]];
	VAR jointtarget SDP_1585 := [[6.36, 36.02, 5.68, 0, 48.31, -223.14], [9E9, 9E9, 9E9, 9E9, 9E9, 9E9]];
	VAR jointtarget SDP_1586 := [[6.09, 35.79, 6.07, 0, 48.14, -232.41], [9E9, 9E9, 9E9, 9E9, 9E9, 9E9]];
	VAR jointtarget SDP_1587 := [[5.79, 35.61, 6.37, 0, 48.02, -241.71], [9E9, 9E9, 9E9, 9E9, 9E9, 9E9]];
	VAR jointtarget SDP_1588 := [[5.47, 35.49, 6.58, 0, 47.93, -251.03], [9E9, 9E9, 9E9, 9E9, 9E9, 9E9]];
	VAR jointtarget SDP_1589 := [[5.13, 35.43, 6.68, 0, 47.89, -260.37], [9E9, 9E9, 9E9, 9E9, 9E9, 9E9]];
	VAR jointtarget SDP_1590 := [[4.05, 35.34, 6.84, 0, 47.82, -265.95], [9E9, 9E9, 9E9, 9E9, 9E9, 9E9]];
	VAR jointtarget SDP_1591 := [[2.97, 35.26, 6.96, 0, 47.77, -267.03], [9E9, 9E9, 9E9, 9E9, 9E9, 9E9]];
	VAR jointtarget SDP_1592 := [[1.89, 35.22, 7.05, 0, 47.74, -268.11], [9E9, 9E9, 9E9, 9E9, 9E9, 9E9]];
	VAR jointtarget SDP_1593 := [[0.8, 35.19, 7.09, 0, 47.72, -269.2], [9E9, 9E9, 9E9, 9E9, 9E9, 9E9]];
	VAR jointtarget SDP_1594 := [[-0.28, 35.18, 7.1, 0, 47.71, -270.28], [9E9, 9E9, 9E9, 9E9, 9E9, 9E9]];
	VAR jointtarget SDP_1595 := [[-1.37, 35.2, 7.07, 0, 47.73, -271.37], [9E9, 9E9, 9E9, 9E9, 9E9, 9E9]];
	VAR jointtarget SDP_1596 := [[-2.45, 35.24, 7.01, 0, 47.75, -272.45], [9E9, 9E9, 9E9, 9E9, 9E9, 9E9]];
	VAR jointtarget SDP_1597 := [[-3.53, 35.3, 6.9, 0, 47.8, -273.53], [9E9, 9E9, 9E9, 9E9, 9E9, 9E9]];
	VAR jointtarget SDP_1598 := [[-4.61, 35.38, 6.76, 0, 47.85, -274.61], [9E9, 9E9, 9E9, 9E9, 9E9, 9E9]];
	VAR jointtarget SDP_1599 := [[-5.69, 35.48, 6.59, 0, 47.93, -275.69], [9E9, 9E9, 9E9, 9E9, 9E9, 9E9]];
	VAR jointtarget SDP_1600 := [[-5.72, 35.49, 6.58, 0, 47.93, -276.38], [9E9, 9E9, 9E9, 9E9, 9E9, 9E9]];
	VAR jointtarget SDP_1601 := [[-5.75, 35.49, 6.57, 0, 47.93, -277.74], [9E9, 9E9, 9E9, 9E9, 9E9, 9E9]];
	VAR jointtarget SDP_1602 := [[-5.79, 35.5, 6.56, 0, 47.94, -279.1], [9E9, 9E9, 9E9, 9E9, 9E9, 9E9]];
	VAR jointtarget SDP_1603 := [[-5.82, 35.51, 6.55, 0, 47.94, -280.46], [9E9, 9E9, 9E9, 9E9, 9E9, 9E9]];
	VAR jointtarget SDP_1604 := [[-5.85, 35.51, 6.54, 0, 47.95, -281.81], [9E9, 9E9, 9E9, 9E9, 9E9, 9E9]];
	VAR jointtarget SDP_1605 := [[-5.89, 35.52, 6.52, 0, 47.95, -283.17], [9E9, 9E9, 9E9, 9E9, 9E9, 9E9]];
	VAR jointtarget SDP_1606 := [[-5.92, 35.53, 6.51, 0, 47.96, -284.53], [9E9, 9E9, 9E9, 9E9, 9E9, 9E9]];
	VAR jointtarget SDP_1607 := [[-5.95, 35.54, 6.49, 0, 47.97, -285.88], [9E9, 9E9, 9E9, 9E9, 9E9, 9E9]];
	VAR jointtarget SDP_1608 := [[-5.98, 35.55, 6.47, 0, 47.98, -287.24], [9E9, 9E9, 9E9, 9E9, 9E9, 9E9]];
	VAR jointtarget SDP_1609 := [[-6.02, 35.56, 6.45, 0, 47.98, -288.59], [9E9, 9E9, 9E9, 9E9, 9E9, 9E9]];
	VAR jointtarget SDP_1610 := [[-6.14, 35.61, 6.37, 0, 48.02, -289.38], [9E9, 9E9, 9E9, 9E9, 9E9, 9E9]];
	VAR jointtarget SDP_1611 := [[-6.27, 35.66, 6.29, 0, 48.05, -289.51], [9E9, 9E9, 9E9, 9E9, 9E9, 9E9]];
	VAR jointtarget SDP_1612 := [[-6.4, 35.71, 6.2, 0, 48.09, -289.64], [9E9, 9E9, 9E9, 9E9, 9E9, 9E9]];
	VAR jointtarget SDP_1613 := [[-6.53, 35.76, 6.12, 0, 48.12, -289.77], [9E9, 9E9, 9E9, 9E9, 9E9, 9E9]];
	VAR jointtarget SDP_1614 := [[-6.66, 35.81, 6.03, 0, 48.16, -289.9], [9E9, 9E9, 9E9, 9E9, 9E9, 9E9]];
	VAR jointtarget SDP_1615 := [[-6.78, 35.86, 5.95, 0, 48.19, -290.02], [9E9, 9E9, 9E9, 9E9, 9E9, 9E9]];
	VAR jointtarget SDP_1616 := [[-6.91, 35.91, 5.86, 0, 48.23, -290.15], [9E9, 9E9, 9E9, 9E9, 9E9, 9E9]];
	VAR jointtarget SDP_1617 := [[-7.04, 35.96, 5.77, 0, 48.27, -290.28], [9E9, 9E9, 9E9, 9E9, 9E9, 9E9]];
	VAR jointtarget SDP_1618 := [[-7.16, 36.01, 5.69, 0, 48.3, -290.4], [9E9, 9E9, 9E9, 9E9, 9E9, 9E9]];
	VAR jointtarget SDP_1619 := [[-7.29, 36.06, 5.6, 0, 48.34, -290.53], [9E9, 9E9, 9E9, 9E9, 9E9, 9E9]];
	VAR jointtarget SDP_1620 := [[-7.55, 36.11, 5.51, 0, 48.38, -280.46], [9E9, 9E9, 9E9, 9E9, 9E9, 9E9]];
	VAR jointtarget SDP_1621 := [[-7.8, 36.06, 5.6, 0, 48.34, -260.07], [9E9, 9E9, 9E9, 9E9, 9E9, 9E9]];
	VAR jointtarget SDP_1622 := [[-8.03, 35.92, 5.84, 0, 48.24, -239.65], [9E9, 9E9, 9E9, 9E9, 9E9, 9E9]];
	VAR jointtarget SDP_1623 := [[-8.2, 35.7, 6.22, 0, 48.08, -219.17], [9E9, 9E9, 9E9, 9E9, 9E9, 9E9]];
	VAR jointtarget SDP_1624 := [[-8.28, 35.43, 6.68, 0, 47.89, -198.6], [9E9, 9E9, 9E9, 9E9, 9E9, 9E9]];
	VAR jointtarget SDP_1625 := [[-8.27, 35.15, 7.16, 0, 47.69, -177.95], [9E9, 9E9, 9E9, 9E9, 9E9, 9E9]];
	VAR jointtarget SDP_1626 := [[-8.17, 34.89, 7.61, 0, 47.51, -157.19], [9E9, 9E9, 9E9, 9E9, 9E9, 9E9]];
	VAR jointtarget SDP_1627 := [[-7.98, 34.68, 7.95, 0, 47.36, -136.36], [9E9, 9E9, 9E9, 9E9, 9E9, 9E9]];
	VAR jointtarget SDP_1628 := [[-7.74, 34.56, 8.16, 0, 47.28, -115.47], [9E9, 9E9, 9E9, 9E9, 9E9, 9E9]];
	VAR jointtarget SDP_1629 := [[-7.47, 34.54, 8.2, 0, 47.26, -94.56], [9E9, 9E9, 9E9, 9E9, 9E9, 9E9]];
	VAR jointtarget SDP_1630 := [[-7.34, 34.55, 8.17, 0, 47.27, -84.1], [9E9, 9E9, 9E9, 9E9, 9E9, 9E9]];
	VAR jointtarget SDP_1631 := [[-7.2, 34.57, 8.15, 0, 47.29, -83.96], [9E9, 9E9, 9E9, 9E9, 9E9, 9E9]];
	VAR jointtarget SDP_1632 := [[-7.06, 34.58, 8.12, 0, 47.3, -83.82], [9E9, 9E9, 9E9, 9E9, 9E9, 9E9]];
	VAR jointtarget SDP_1633 := [[-6.92, 34.6, 8.09, 0, 47.31, -83.68], [9E9, 9E9, 9E9, 9E9, 9E9, 9E9]];
	VAR jointtarget SDP_1634 := [[-6.79, 34.61, 8.07, 0, 47.32, -83.55], [9E9, 9E9, 9E9, 9E9, 9E9, 9E9]];
	VAR jointtarget SDP_1635 := [[-6.65, 34.63, 8.04, 0, 47.34, -83.41], [9E9, 9E9, 9E9, 9E9, 9E9, 9E9]];
	VAR jointtarget SDP_1636 := [[-6.51, 34.64, 8.01, 0, 47.35, -83.27], [9E9, 9E9, 9E9, 9E9, 9E9, 9E9]];
	VAR jointtarget SDP_1637 := [[-6.38, 34.66, 7.98, 0, 47.36, -83.14], [9E9, 9E9, 9E9, 9E9, 9E9, 9E9]];
	VAR jointtarget SDP_1638 := [[-6.24, 34.67, 7.95, 0, 47.38, -83], [9E9, 9E9, 9E9, 9E9, 9E9, 9E9]];
	VAR jointtarget SDP_1639 := [[-6.1, 34.69, 7.92, 0, 47.39, -82.86], [9E9, 9E9, 9E9, 9E9, 9E9, 9E9]];
	VAR jointtarget SDP_1640 := [[-6.07, 34.69, 7.91, 0, 47.39, -83.49], [9E9, 9E9, 9E9, 9E9, 9E9, 9E9]];
	VAR jointtarget SDP_1641 := [[-6.03, 34.7, 7.91, 0, 47.4, -84.78], [9E9, 9E9, 9E9, 9E9, 9E9, 9E9]];
	VAR jointtarget SDP_1642 := [[-6, 34.7, 7.9, 0, 47.4, -86.07], [9E9, 9E9, 9E9, 9E9, 9E9, 9E9]];
	VAR jointtarget SDP_1643 := [[-5.97, 34.7, 7.9, 0, 47.4, -87.36], [9E9, 9E9, 9E9, 9E9, 9E9, 9E9]];
	VAR jointtarget SDP_1644 := [[-5.93, 34.7, 7.9, 0, 47.4, -88.65], [9E9, 9E9, 9E9, 9E9, 9E9, 9E9]];
	VAR jointtarget SDP_1645 := [[-5.9, 34.7, 7.9, 0, 47.4, -89.94], [9E9, 9E9, 9E9, 9E9, 9E9, 9E9]];
	VAR jointtarget SDP_1646 := [[-5.86, 34.7, 7.9, 0, 47.4, -91.23], [9E9, 9E9, 9E9, 9E9, 9E9, 9E9]];
	VAR jointtarget SDP_1647 := [[-5.83, 34.7, 7.9, 0, 47.4, -92.52], [9E9, 9E9, 9E9, 9E9, 9E9, 9E9]];
	VAR jointtarget SDP_1648 := [[-5.79, 34.7, 7.91, 0, 47.4, -93.81], [9E9, 9E9, 9E9, 9E9, 9E9, 9E9]];
	VAR jointtarget SDP_1649 := [[-5.76, 34.69, 7.91, 0, 47.4, -95.1], [9E9, 9E9, 9E9, 9E9, 9E9, 9E9]];
	VAR jointtarget SDP_1650 := [[-4.6, 34.58, 8.1, 0, 47.32, -94.6], [9E9, 9E9, 9E9, 9E9, 9E9, 9E9]];
	VAR jointtarget SDP_1651 := [[-3.43, 34.5, 8.25, 0, 47.26, -93.43], [9E9, 9E9, 9E9, 9E9, 9E9, 9E9]];
	VAR jointtarget SDP_1652 := [[-2.26, 34.44, 8.35, 0, 47.22, -92.26], [9E9, 9E9, 9E9, 9E9, 9E9, 9E9]];
	VAR jointtarget SDP_1653 := [[-1.09, 34.4, 8.41, 0, 47.19, -91.09], [9E9, 9E9, 9E9, 9E9, 9E9, 9E9]];
	VAR jointtarget SDP_1654 := [[0.09, 34.39, 8.43, 0, 47.18, -89.91], [9E9, 9E9, 9E9, 9E9, 9E9, 9E9]];
	VAR jointtarget SDP_1655 := [[1.26, 34.4, 8.4, 0, 47.19, -88.74], [9E9, 9E9, 9E9, 9E9, 9E9, 9E9]];
	VAR jointtarget SDP_1656 := [[2.43, 34.44, 8.34, 0, 47.22, -87.57], [9E9, 9E9, 9E9, 9E9, 9E9, 9E9]];
	VAR jointtarget SDP_1657 := [[3.6, 34.51, 8.23, 0, 47.27, -86.4], [9E9, 9E9, 9E9, 9E9, 9E9, 9E9]];
	VAR jointtarget SDP_1658 := [[4.77, 34.6, 8.07, 0, 47.33, -85.23], [9E9, 9E9, 9E9, 9E9, 9E9, 9E9]];
	VAR jointtarget SDP_1659 := [[5.93, 34.71, 7.88, 0, 47.41, -84.07], [9E9, 9E9, 9E9, 9E9, 9E9, 9E9]];
	VAR jointtarget SDP_1660 := [[6.27, 34.78, 7.76, 0, 47.46, -79.23], [9E9, 9E9, 9E9, 9E9, 9E9, 9E9]];
	VAR jointtarget SDP_1661 := [[6.6, 34.9, 7.55, 0, 47.54, -69.9], [9E9, 9E9, 9E9, 9E9, 9E9, 9E9]];
	VAR jointtarget SDP_1662 := [[6.9, 35.08, 7.25, 0, 47.67, -60.6], [9E9, 9E9, 9E9, 9E9, 9E9, 9E9]];
	VAR jointtarget SDP_1663 := [[7.17, 35.31, 6.85, 0, 47.83, -51.33], [9E9, 9E9, 9E9, 9E9, 9E9, 9E9]];
	VAR jointtarget SDP_1664 := [[7.4, 35.59, 6.39, 0, 48.03, -42.1], [9E9, 9E9, 9E9, 9E9, 9E9, 9E9]];
	VAR jointtarget SDP_1665 := [[7.59, 35.9, 5.86, 0, 48.25, -32.91], [9E9, 9E9, 9E9, 9E9, 9E9, 9E9]];
	VAR jointtarget SDP_1666 := [[7.73, 36.24, 5.27, 0, 48.49, -23.77], [9E9, 9E9, 9E9, 9E9, 9E9, 9E9]];
	VAR jointtarget SDP_1667 := [[7.82, 36.6, 4.65, 0, 48.75, -14.68], [9E9, 9E9, 9E9, 9E9, 9E9, 9E9]];
	VAR jointtarget SDP_1668 := [[7.85, 36.97, 4.02, 0, 49.02, -5.65], [9E9, 9E9, 9E9, 9E9, 9E9, 9E9]];
	VAR jointtarget SDP_1669 := [[7.83, 37.34, 3.37, 0, 49.29, 3.33], [9E9, 9E9, 9E9, 9E9, 9E9, 9E9]];
	VAR jointtarget SDP_1670 := [[7.68, 38.6, 1.2, 0, 50.2, 7.68], [9E9, 9E9, 9E9, 9E9, 9E9, 9E9]];
	VAR jointtarget SDP_1671 := [[7.54, 39.87, -1.02, 0, 51.15, 7.54], [9E9, 9E9, 9E9, 9E9, 9E9, 9E9]];
	VAR jointtarget SDP_1672 := [[7.4, 41.16, -3.28, 0, 52.12, 7.4], [9E9, 9E9, 9E9, 9E9, 9E9, 9E9]];
	VAR jointtarget SDP_1673 := [[7.26, 42.47, -5.59, 0, 53.12, 7.26], [9E9, 9E9, 9E9, 9E9, 9E9, 9E9]];
	VAR jointtarget SDP_1674 := [[7.13, 43.8, -7.96, 0, 54.15, 7.13], [9E9, 9E9, 9E9, 9E9, 9E9, 9E9]];
	VAR jointtarget SDP_1675 := [[7.01, 45.17, -10.39, 0, 55.22, 7.01], [9E9, 9E9, 9E9, 9E9, 9E9, 9E9]];
	VAR jointtarget SDP_1676 := [[6.89, 46.56, -12.88, 0, 56.32, 6.89], [9E9, 9E9, 9E9, 9E9, 9E9, 9E9]];
	VAR jointtarget SDP_1677 := [[6.77, 47.98, -15.45, 0, 57.47, 6.77], [9E9, 9E9, 9E9, 9E9, 9E9, 9E9]];
	VAR jointtarget SDP_1678 := [[6.66, 49.45, -18.1, 0, 58.65, 6.66], [9E9, 9E9, 9E9, 9E9, 9E9, 9E9]];
	VAR jointtarget SDP_1679 := [[6.55, 50.96, -20.84, 0, 59.88, 6.55], [9E9, 9E9, 9E9, 9E9, 9E9, 9E9]];
	VAR jointtarget SDP_1680 := [[6.55, 51, -20.92, 0, 59.92, 5.89], [9E9, 9E9, 9E9, 9E9, 9E9, 9E9]];
	VAR jointtarget SDP_1681 := [[6.55, 51.05, -21, 0, 59.96, 4.56], [9E9, 9E9, 9E9, 9E9, 9E9, 9E9]];
	VAR jointtarget SDP_1682 := [[6.55, 51.09, -21.09, 0, 60, 3.24], [9E9, 9E9, 9E9, 9E9, 9E9, 9E9]];
	VAR jointtarget SDP_1683 := [[6.54, 51.14, -21.17, 0, 60.03, 1.91], [9E9, 9E9, 9E9, 9E9, 9E9, 9E9]];
	VAR jointtarget SDP_1684 := [[6.54, 51.18, -21.25, 0, 60.07, 0.59], [9E9, 9E9, 9E9, 9E9, 9E9, 9E9]];
	VAR jointtarget SDP_1685 := [[6.54, 51.23, -21.34, 0, 60.11, -0.74], [9E9, 9E9, 9E9, 9E9, 9E9, 9E9]];
	VAR jointtarget SDP_1686 := [[6.55, 51.27, -21.42, 0, 60.14, -2.06], [9E9, 9E9, 9E9, 9E9, 9E9, 9E9]];
	VAR jointtarget SDP_1687 := [[6.55, 51.32, -21.5, 0, 60.18, -3.38], [9E9, 9E9, 9E9, 9E9, 9E9, 9E9]];
	VAR jointtarget SDP_1688 := [[6.55, 51.36, -21.58, 0, 60.22, -4.7], [9E9, 9E9, 9E9, 9E9, 9E9, 9E9]];
	VAR jointtarget SDP_1689 := [[6.55, 51.41, -21.67, 0, 60.26, -6.03], [9E9, 9E9, 9E9, 9E9, 9E9, 9E9]];
	VAR jointtarget SDP_1690 := [[6.57, 51.59, -22, 0, 60.41, -6.68], [9E9, 9E9, 9E9, 9E9, 9E9, 9E9]];
	VAR jointtarget SDP_1691 := [[6.58, 51.78, -22.34, 0, 60.56, -6.66], [9E9, 9E9, 9E9, 9E9, 9E9, 9E9]];
	VAR jointtarget SDP_1692 := [[6.59, 51.96, -22.67, 0, 60.71, -6.65], [9E9, 9E9, 9E9, 9E9, 9E9, 9E9]];
	VAR jointtarget SDP_1693 := [[6.6, 52.15, -23.01, 0, 60.87, -6.64], [9E9, 9E9, 9E9, 9E9, 9E9, 9E9]];
	VAR jointtarget SDP_1694 := [[6.62, 52.33, -23.35, 0, 61.02, -6.62], [9E9, 9E9, 9E9, 9E9, 9E9, 9E9]];
	VAR jointtarget SDP_1695 := [[6.63, 52.52, -23.69, 0, 61.18, -6.61], [9E9, 9E9, 9E9, 9E9, 9E9, 9E9]];
	VAR jointtarget SDP_1696 := [[6.64, 52.71, -24.04, 0, 61.33, -6.6], [9E9, 9E9, 9E9, 9E9, 9E9, 9E9]];
	VAR jointtarget SDP_1697 := [[6.65, 52.9, -24.38, 0, 61.49, -6.59], [9E9, 9E9, 9E9, 9E9, 9E9, 9E9]];
	VAR jointtarget SDP_1698 := [[6.67, 53.08, -24.73, 0, 61.65, -6.57], [9E9, 9E9, 9E9, 9E9, 9E9, 9E9]];
	VAR jointtarget SDP_1699 := [[6.68, 53.27, -25.08, 0, 61.8, -6.56], [9E9, 9E9, 9E9, 9E9, 9E9, 9E9]];
	VAR jointtarget SDP_1700 := [[6.66, 53.65, -25.76, 0, 62.11, 3.75], [9E9, 9E9, 9E9, 9E9, 9E9, 9E9]];
	VAR jointtarget SDP_1701 := [[6.58, 53.99, -26.39, 0, 62.4, 24.31], [9E9, 9E9, 9E9, 9E9, 9E9, 9E9]];
	VAR jointtarget SDP_1702 := [[6.43, 54.26, -26.89, 0, 62.63, 44.81], [9E9, 9E9, 9E9, 9E9, 9E9, 9E9]];
	VAR jointtarget SDP_1703 := [[6.24, 54.42, -27.18, 0, 62.76, 65.27], [9E9, 9E9, 9E9, 9E9, 9E9, 9E9]];
	VAR jointtarget SDP_1704 := [[6.04, 54.45, -27.23, 0, 62.78, 85.71], [9E9, 9E9, 9E9, 9E9, 9E9, 9E9]];
	VAR jointtarget SDP_1705 := [[5.84, 54.34, -27.03, 0, 62.69, 106.16], [9E9, 9E9, 9E9, 9E9, 9E9, 9E9]];
	VAR jointtarget SDP_1706 := [[5.67, 54.11, -26.61, 0, 62.5, 126.64], [9E9, 9E9, 9E9, 9E9, 9E9, 9E9]];
	VAR jointtarget SDP_1707 := [[5.56, 53.79, -26.03, 0, 62.24, 147.18], [9E9, 9E9, 9E9, 9E9, 9E9, 9E9]];
	VAR jointtarget SDP_1708 := [[5.52, 53.43, -25.36, 0, 61.93, 167.78], [9E9, 9E9, 9E9, 9E9, 9E9, 9E9]];
	VAR jointtarget SDP_1709 := [[5.55, 53.06, -24.69, 0, 61.63, 188.46], [9E9, 9E9, 9E9, 9E9, 9E9, 9E9]];
	VAR jointtarget SDP_1710 := [[5.58, 52.88, -24.36, 0, 61.48, 198.82], [9E9, 9E9, 9E9, 9E9, 9E9, 9E9]];
	VAR jointtarget SDP_1711 := [[5.62, 52.7, -24.03, 0, 61.33, 198.86], [9E9, 9E9, 9E9, 9E9, 9E9, 9E9]];
	VAR jointtarget SDP_1712 := [[5.65, 52.52, -23.7, 0, 61.18, 198.89], [9E9, 9E9, 9E9, 9E9, 9E9, 9E9]];
	VAR jointtarget SDP_1713 := [[5.69, 52.34, -23.37, 0, 61.03, 198.93], [9E9, 9E9, 9E9, 9E9, 9E9, 9E9]];
	VAR jointtarget SDP_1714 := [[5.72, 52.17, -23.05, 0, 60.88, 198.96], [9E9, 9E9, 9E9, 9E9, 9E9, 9E9]];
	VAR jointtarget SDP_1715 := [[5.76, 51.99, -22.73, 0, 60.74, 199], [9E9, 9E9, 9E9, 9E9, 9E9, 9E9]];
	VAR jointtarget SDP_1716 := [[5.79, 51.81, -22.41, 0, 60.59, 199.03], [9E9, 9E9, 9E9, 9E9, 9E9, 9E9]];
	VAR jointtarget SDP_1717 := [[5.83, 51.64, -22.09, 0, 60.45, 199.07], [9E9, 9E9, 9E9, 9E9, 9E9, 9E9]];
	VAR jointtarget SDP_1718 := [[5.87, 51.46, -21.77, 0, 60.3, 199.11], [9E9, 9E9, 9E9, 9E9, 9E9, 9E9]];
	VAR jointtarget SDP_1719 := [[5.9, 51.29, -21.45, 0, 60.16, 199.14], [9E9, 9E9, 9E9, 9E9, 9E9, 9E9]];
	VAR jointtarget SDP_1720 := [[5.91, 51.25, -21.37, 0, 60.12, 198.49], [9E9, 9E9, 9E9, 9E9, 9E9, 9E9]];
	VAR jointtarget SDP_1721 := [[5.92, 51.2, -21.29, 0, 60.09, 197.17], [9E9, 9E9, 9E9, 9E9, 9E9, 9E9]];
	VAR jointtarget SDP_1722 := [[5.93, 51.16, -21.21, 0, 60.05, 195.86], [9E9, 9E9, 9E9, 9E9, 9E9, 9E9]];
	VAR jointtarget SDP_1723 := [[5.93, 51.12, -21.13, 0, 60.02, 194.54], [9E9, 9E9, 9E9, 9E9, 9E9, 9E9]];
	VAR jointtarget SDP_1724 := [[5.94, 51.07, -21.05, 0, 59.98, 193.22], [9E9, 9E9, 9E9, 9E9, 9E9, 9E9]];
	VAR jointtarget SDP_1725 := [[5.94, 51.03, -20.97, 0, 59.94, 191.9], [9E9, 9E9, 9E9, 9E9, 9E9, 9E9]];
	VAR jointtarget SDP_1726 := [[5.95, 50.98, -20.89, 0, 59.91, 190.58], [9E9, 9E9, 9E9, 9E9, 9E9, 9E9]];
	VAR jointtarget SDP_1727 := [[5.95, 50.94, -20.81, 0, 59.87, 189.26], [9E9, 9E9, 9E9, 9E9, 9E9, 9E9]];
	VAR jointtarget SDP_1728 := [[5.96, 50.89, -20.73, 0, 59.83, 187.94], [9E9, 9E9, 9E9, 9E9, 9E9, 9E9]];
	VAR jointtarget SDP_1729 := [[5.96, 50.85, -20.65, 0, 59.8, 186.62], [9E9, 9E9, 9E9, 9E9, 9E9, 9E9]];
	VAR jointtarget SDP_1730 := [[6.05, 49.44, -18.08, 0, 58.64, 186.05], [9E9, 9E9, 9E9, 9E9, 9E9, 9E9]];
	VAR jointtarget SDP_1731 := [[6.15, 48.06, -15.59, 0, 57.53, 186.15], [9E9, 9E9, 9E9, 9E9, 9E9, 9E9]];
	VAR jointtarget SDP_1732 := [[6.25, 46.72, -13.18, 0, 56.45, 186.25], [9E9, 9E9, 9E9, 9E9, 9E9, 9E9]];
	VAR jointtarget SDP_1733 := [[6.35, 45.41, -10.83, 0, 55.42, 186.35], [9E9, 9E9, 9E9, 9E9, 9E9, 9E9]];
	VAR jointtarget SDP_1734 := [[6.46, 44.13, -8.54, 0, 54.41, 186.46], [9E9, 9E9, 9E9, 9E9, 9E9, 9E9]];
	VAR jointtarget SDP_1735 := [[6.56, 42.87, -6.3, 0, 53.43, 186.56], [9E9, 9E9, 9E9, 9E9, 9E9, 9E9]];
	VAR jointtarget SDP_1736 := [[6.68, 41.64, -4.12, 0, 52.48, 186.68], [9E9, 9E9, 9E9, 9E9, 9E9, 9E9]];
	VAR jointtarget SDP_1737 := [[6.79, 40.42, -1.98, 0, 51.56, 186.79], [9E9, 9E9, 9E9, 9E9, 9E9, 9E9]];
	VAR jointtarget SDP_1738 := [[6.91, 39.22, 0.12, 0, 50.66, 186.91], [9E9, 9E9, 9E9, 9E9, 9E9, 9E9]];
	VAR jointtarget SDP_1739 := [[7.04, 38.03, 2.18, 0, 49.79, 187.04], [9E9, 9E9, 9E9, 9E9, 9E9, 9E9]];
	VAR jointtarget SDP_1740 := [[7.05, 37.66, 2.83, 0, 49.51, 182.55], [9E9, 9E9, 9E9, 9E9, 9E9, 9E9]];
	VAR jointtarget SDP_1741 := [[7.02, 37.28, 3.47, 0, 49.24, 173.52], [9E9, 9E9, 9E9, 9E9, 9E9, 9E9]];
	VAR jointtarget SDP_1742 := [[6.93, 36.92, 4.1, 0, 48.98, 164.43], [9E9, 9E9, 9E9, 9E9, 9E9, 9E9]];
	VAR jointtarget SDP_1743 := [[6.78, 36.58, 4.68, 0, 48.74, 155.28], [9E9, 9E9, 9E9, 9E9, 9E9, 9E9]];
	VAR jointtarget SDP_1744 := [[6.6, 36.27, 5.21, 0, 48.51, 146.1], [9E9, 9E9, 9E9, 9E9, 9E9, 9E9]];
	VAR jointtarget SDP_1745 := [[6.36, 36, 5.68, 0, 48.32, 136.86], [9E9, 9E9, 9E9, 9E9, 9E9, 9E9]];
	VAR jointtarget SDP_1746 := [[6.09, 35.78, 6.07, 0, 48.16, 127.59], [9E9, 9E9, 9E9, 9E9, 9E9, 9E9]];
	VAR jointtarget SDP_1747 := [[5.79, 35.6, 6.37, 0, 48.03, 118.29], [9E9, 9E9, 9E9, 9E9, 9E9, 9E9]];
	VAR jointtarget SDP_1748 := [[5.47, 35.48, 6.57, 0, 47.95, 108.97], [9E9, 9E9, 9E9, 9E9, 9E9, 9E9]];
	VAR jointtarget SDP_1749 := [[5.13, 35.41, 6.68, 0, 47.9, 99.63], [9E9, 9E9, 9E9, 9E9, 9E9, 9E9]];
	VAR jointtarget SDP_1750 := [[4.07, 35.32, 6.84, 0, 47.84, 94.07], [9E9, 9E9, 9E9, 9E9, 9E9, 9E9]];
	VAR jointtarget SDP_1751 := [[3.01, 35.25, 6.96, 0, 47.79, 93.01], [9E9, 9E9, 9E9, 9E9, 9E9, 9E9]];
	VAR jointtarget SDP_1752 := [[1.95, 35.2, 7.04, 0, 47.76, 91.95], [9E9, 9E9, 9E9, 9E9, 9E9, 9E9]];
	VAR jointtarget SDP_1753 := [[0.89, 35.18, 7.09, 0, 47.74, 90.89], [9E9, 9E9, 9E9, 9E9, 9E9, 9E9]];
	VAR jointtarget SDP_1754 := [[-0.18, 35.17, 7.1, 0, 47.73, 89.82], [9E9, 9E9, 9E9, 9E9, 9E9, 9E9]];
	VAR jointtarget SDP_1755 := [[-1.24, 35.18, 7.08, 0, 47.74, 88.76], [9E9, 9E9, 9E9, 9E9, 9E9, 9E9]];
	VAR jointtarget SDP_1756 := [[-2.31, 35.22, 7.02, 0, 47.77, 87.69], [9E9, 9E9, 9E9, 9E9, 9E9, 9E9]];
	VAR jointtarget SDP_1757 := [[-3.37, 35.27, 6.92, 0, 47.8, 86.63], [9E9, 9E9, 9E9, 9E9, 9E9, 9E9]];
	VAR jointtarget SDP_1758 := [[-4.43, 35.35, 6.79, 0, 47.86, 85.57], [9E9, 9E9, 9E9, 9E9, 9E9, 9E9]];
	VAR jointtarget SDP_1759 := [[-5.48, 35.45, 6.62, 0, 47.93, 84.52], [9E9, 9E9, 9E9, 9E9, 9E9, 9E9]];
	VAR jointtarget SDP_1760 := [[-5.59, 35.46, 6.61, 0, 47.93, 86.6], [9E9, 9E9, 9E9, 9E9, 9E9, 9E9]];
	VAR jointtarget SDP_1761 := [[-5.71, 35.46, 6.61, 0, 47.93, 90.88], [9E9, 9E9, 9E9, 9E9, 9E9, 9E9]];
	VAR jointtarget SDP_1762 := [[-5.82, 35.44, 6.63, 0, 47.92, 95.15], [9E9, 9E9, 9E9, 9E9, 9E9, 9E9]];
	VAR jointtarget SDP_1763 := [[-5.93, 35.42, 6.66, 0, 47.91, 99.43], [9E9, 9E9, 9E9, 9E9, 9E9, 9E9]];
	VAR jointtarget SDP_1764 := [[-6.04, 35.4, 6.71, 0, 47.89, 103.71], [9E9, 9E9, 9E9, 9E9, 9E9, 9E9]];
	VAR jointtarget SDP_1765 := [[-6.14, 35.36, 6.78, 0, 47.86, 107.99], [9E9, 9E9, 9E9, 9E9, 9E9, 9E9]];
	VAR jointtarget SDP_1766 := [[-6.25, 35.31, 6.86, 0, 47.83, 112.27], [9E9, 9E9, 9E9, 9E9, 9E9, 9E9]];
	VAR jointtarget SDP_1767 := [[-6.35, 35.26, 6.95, 0, 47.79, 116.56], [9E9, 9E9, 9E9, 9E9, 9E9, 9E9]];
	VAR jointtarget SDP_1768 := [[-6.44, 35.2, 7.05, 0, 47.75, 120.85], [9E9, 9E9, 9E9, 9E9, 9E9, 9E9]];
	VAR jointtarget SDP_1769 := [[-6.54, 35.13, 7.17, 0, 47.7, 125.15], [9E9, 9E9, 9E9, 9E9, 9E9, 9E9]];
	VAR jointtarget SDP_1770 := [[-6.59, 35.08, 7.24, 0, 47.67, 127.29], [9E9, 9E9, 9E9, 9E9, 9E9, 9E9]];
	VAR jointtarget SDP_1771 := [[-6.64, 35.04, 7.32, 0, 47.64, 127.23], [9E9, 9E9, 9E9, 9E9, 9E9, 9E9]];
	VAR jointtarget SDP_1772 := [[-6.7, 35, 7.39, 0, 47.61, 127.18], [9E9, 9E9, 9E9, 9E9, 9E9, 9E9]];
	VAR jointtarget SDP_1773 := [[-6.75, 34.95, 7.47, 0, 47.58, 127.12], [9E9, 9E9, 9E9, 9E9, 9E9, 9E9]];
	VAR jointtarget SDP_1774 := [[-6.81, 34.91, 7.54, 0, 47.55, 127.07], [9E9, 9E9, 9E9, 9E9, 9E9, 9E9]];
	VAR jointtarget SDP_1775 := [[-6.86, 34.87, 7.62, 0, 47.52, 127.01], [9E9, 9E9, 9E9, 9E9, 9E9, 9E9]];
	VAR jointtarget SDP_1776 := [[-6.92, 34.82, 7.69, 0, 47.49, 126.96], [9E9, 9E9, 9E9, 9E9, 9E9, 9E9]];
	VAR jointtarget SDP_1777 := [[-6.97, 34.78, 7.76, 0, 47.46, 126.91], [9E9, 9E9, 9E9, 9E9, 9E9, 9E9]];
	VAR jointtarget SDP_1778 := [[-7.03, 34.74, 7.84, 0, 47.43, 126.85], [9E9, 9E9, 9E9, 9E9, 9E9, 9E9]];
	VAR jointtarget SDP_1779 := [[-7.08, 34.69, 7.91, 0, 47.4, 126.8], [9E9, 9E9, 9E9, 9E9, 9E9, 9E9]];
	VAR jointtarget SDP_1780 := [[-7.39, 34.55, 8.15, 0, 47.3, 113.1], [9E9, 9E9, 9E9, 9E9, 9E9, 9E9]];
	VAR jointtarget SDP_1781 := [[-7.72, 34.58, 8.11, 0, 47.31, 85.99], [9E9, 9E9, 9E9, 9E9, 9E9, 9E9]];
	VAR jointtarget SDP_1782 := [[-8.01, 34.76, 7.8, 0, 47.44, 58.93], [9E9, 9E9, 9E9, 9E9, 9E9, 9E9]];
	VAR jointtarget SDP_1783 := [[-8.18, 35.06, 7.29, 0, 47.65, 31.98], [9E9, 9E9, 9E9, 9E9, 9E9, 9E9]];
	VAR jointtarget SDP_1784 := [[-8.21, 35.41, 6.7, 0, 47.9, 5.18], [9E9, 9E9, 9E9, 9E9, 9E9, 9E9]];
	VAR jointtarget SDP_1785 := [[-8.09, 35.74, 6.13, 0, 48.13, -21.48], [9E9, 9E9, 9E9, 9E9, 9E9, 9E9]];
	VAR jointtarget SDP_1786 := [[-7.85, 35.97, 5.73, 0, 48.3, -48.01], [9E9, 9E9, 9E9, 9E9, 9E9, 9E9]];
	VAR jointtarget SDP_1787 := [[-7.53, 36.07, 5.57, 0, 48.37, -74.47], [9E9, 9E9, 9E9, 9E9, 9E9, 9E9]];
	VAR jointtarget SDP_1788 := [[-7.21, 36, 5.69, 0, 48.32, -100.93], [9E9, 9E9, 9E9, 9E9, 9E9, 9E9]];
	VAR jointtarget SDP_1789 := [[-6.96, 35.78, 6.06, 0, 48.16, -127.44], [9E9, 9E9, 9E9, 9E9, 9E9, 9E9]];
	VAR jointtarget SDP_1790 := [[-6.9, 35.71, 6.18, 0, 48.11, -140.78], [9E9, 9E9, 9E9, 9E9, 9E9, 9E9]];
	VAR jointtarget SDP_1791 := [[-6.85, 35.64, 6.3, 0, 48.06, -140.72], [9E9, 9E9, 9E9, 9E9, 9E9, 9E9]];
	VAR jointtarget SDP_1792 := [[-6.79, 35.57, 6.42, 0, 48.01, -140.67], [9E9, 9E9, 9E9, 9E9, 9E9, 9E9]];
	VAR jointtarget SDP_1793 := [[-6.74, 35.5, 6.54, 0, 47.96, -140.62], [9E9, 9E9, 9E9, 9E9, 9E9, 9E9]];
	VAR jointtarget SDP_1794 := [[-6.68, 35.42, 6.66, 0, 47.91, -140.56], [9E9, 9E9, 9E9, 9E9, 9E9, 9E9]];
	VAR jointtarget SDP_1795 := [[-6.63, 35.35, 6.79, 0, 47.86, -140.51], [9E9, 9E9, 9E9, 9E9, 9E9, 9E9]];
	VAR jointtarget SDP_1796 := [[-6.58, 35.28, 6.91, 0, 47.81, -140.45], [9E9, 9E9, 9E9, 9E9, 9E9, 9E9]];
	VAR jointtarget SDP_1797 := [[-6.52, 35.21, 7.03, 0, 47.76, -140.4], [9E9, 9E9, 9E9, 9E9, 9E9, 9E9]];
	VAR jointtarget SDP_1798 := [[-6.47, 35.14, 7.15, 0, 47.71, -140.34], [9E9, 9E9, 9E9, 9E9, 9E9, 9E9]];
	VAR jointtarget SDP_1799 := [[-6.41, 35.07, 7.27, 0, 47.66, -140.29], [9E9, 9E9, 9E9, 9E9, 9E9, 9E9]];
	VAR jointtarget SDP_1800 := [[-6.38, 35.04, 7.32, 0, 47.64, -139.16], [9E9, 9E9, 9E9, 9E9, 9E9, 9E9]];
	VAR jointtarget SDP_1801 := [[-6.36, 35.01, 7.37, 0, 47.62, -136.92], [9E9, 9E9, 9E9, 9E9, 9E9, 9E9]];
	VAR jointtarget SDP_1802 := [[-6.33, 34.98, 7.42, 0, 47.6, -134.69], [9E9, 9E9, 9E9, 9E9, 9E9, 9E9]];
	VAR jointtarget SDP_1803 := [[-6.3, 34.95, 7.47, 0, 47.58, -132.45], [9E9, 9E9, 9E9, 9E9, 9E9, 9E9]];
	VAR jointtarget SDP_1804 := [[-6.27, 34.92, 7.52, 0, 47.56, -130.22], [9E9, 9E9, 9E9, 9E9, 9E9, 9E9]];
	VAR jointtarget SDP_1805 := [[-6.24, 34.9, 7.56, 0, 47.54, -127.98], [9E9, 9E9, 9E9, 9E9, 9E9, 9E9]];
	VAR jointtarget SDP_1806 := [[-6.21, 34.87, 7.6, 0, 47.53, -125.74], [9E9, 9E9, 9E9, 9E9, 9E9, 9E9]];
	VAR jointtarget SDP_1807 := [[-6.18, 34.85, 7.64, 0, 47.51, -123.5], [9E9, 9E9, 9E9, 9E9, 9E9, 9E9]];
	VAR jointtarget SDP_1808 := [[-6.14, 34.82, 7.68, 0, 47.5, -121.26], [9E9, 9E9, 9E9, 9E9, 9E9, 9E9]];
	VAR jointtarget SDP_1809 := [[-6.11, 34.8, 7.71, 0, 47.49, -119.01], [9E9, 9E9, 9E9, 9E9, 9E9, 9E9]];
	VAR jointtarget SDP_1810 := [[-6.09, 34.79, 7.73, 0, 47.48, -117.89], [9E9, 9E9, 9E9, 9E9, 9E9, 9E9]];
	VAR jointtarget SDP_1811 := [[-6.07, 34.78, 7.74, 0, 47.47, -117.87], [9E9, 9E9, 9E9, 9E9, 9E9, 9E9]];
	VAR jointtarget SDP_1812 := [[-6.05, 34.77, 7.76, 0, 47.47, -117.86], [9E9, 9E9, 9E9, 9E9, 9E9, 9E9]];
	VAR jointtarget SDP_1813 := [[-6.04, 34.76, 7.78, 0, 47.46, -117.84], [9E9, 9E9, 9E9, 9E9, 9E9, 9E9]];
	VAR jointtarget SDP_1814 := [[-6.02, 34.75, 7.79, 0, 47.45, -117.82], [9E9, 9E9, 9E9, 9E9, 9E9, 9E9]];
	VAR jointtarget SDP_1815 := [[-6, 34.74, 7.81, 0, 47.45, -117.8], [9E9, 9E9, 9E9, 9E9, 9E9, 9E9]];
	VAR jointtarget SDP_1816 := [[-5.98, 34.73, 7.83, 0, 47.44, -117.79], [9E9, 9E9, 9E9, 9E9, 9E9, 9E9]];
	VAR jointtarget SDP_1817 := [[-5.97, 34.72, 7.84, 0, 47.44, -117.77], [9E9, 9E9, 9E9, 9E9, 9E9, 9E9]];
	VAR jointtarget SDP_1818 := [[-5.95, 34.71, 7.86, 0, 47.43, -117.75], [9E9, 9E9, 9E9, 9E9, 9E9, 9E9]];
	VAR jointtarget SDP_1819 := [[-5.93, 34.7, 7.88, 0, 47.42, -117.73], [9E9, 9E9, 9E9, 9E9, 9E9, 9E9]];
	VAR jointtarget SDP_1820 := [[-4.75, 34.58, 8.07, 0, 47.34, -94.75], [9E9, 9E9, 9E9, 9E9, 9E9, 9E9]];
	VAR jointtarget SDP_1821 := [[-3.57, 34.49, 8.23, 0, 47.28, -93.57], [9E9, 9E9, 9E9, 9E9, 9E9, 9E9]];
	VAR jointtarget SDP_1822 := [[-2.38, 34.43, 8.34, 0, 47.23, -92.38], [9E9, 9E9, 9E9, 9E9, 9E9, 9E9]];
	VAR jointtarget SDP_1823 := [[-1.19, 34.39, 8.4, 0, 47.21, -91.19], [9E9, 9E9, 9E9, 9E9, 9E9, 9E9]];
	VAR jointtarget SDP_1824 := [[0, 34.38, 8.43, 0, 47.2, -90], [9E9, 9E9, 9E9, 9E9, 9E9, 9E9]];
	VAR jointtarget SDP_1825 := [[1.19, 34.39, 8.4, 0, 47.21, -88.81], [9E9, 9E9, 9E9, 9E9, 9E9, 9E9]];
	VAR jointtarget SDP_1826 := [[2.38, 34.43, 8.34, 0, 47.23, -87.62], [9E9, 9E9, 9E9, 9E9, 9E9, 9E9]];
	VAR jointtarget SDP_1827 := [[3.57, 34.49, 8.23, 0, 47.28, -86.43], [9E9, 9E9, 9E9, 9E9, 9E9, 9E9]];
	VAR jointtarget SDP_1828 := [[4.75, 34.58, 8.07, 0, 47.34, -85.25], [9E9, 9E9, 9E9, 9E9, 9E9, 9E9]];
	VAR jointtarget SDP_1829 := [[5.93, 34.7, 7.88, 0, 47.42, -84.07], [9E9, 9E9, 9E9, 9E9, 9E9, 9E9]];
	VAR jointtarget SDP_1830 := [[6.27, 34.77, 7.76, 0, 47.47, -79.23], [9E9, 9E9, 9E9, 9E9, 9E9, 9E9]];
	VAR jointtarget SDP_1831 := [[6.6, 34.89, 7.55, 0, 47.56, -69.9], [9E9, 9E9, 9E9, 9E9, 9E9, 9E9]];
	VAR jointtarget SDP_1832 := [[6.9, 35.07, 7.24, 0, 47.69, -60.6], [9E9, 9E9, 9E9, 9E9, 9E9, 9E9]];
	VAR jointtarget SDP_1833 := [[7.17, 35.3, 6.85, 0, 47.85, -51.33], [9E9, 9E9, 9E9, 9E9, 9E9, 9E9]];
	VAR jointtarget SDP_1834 := [[7.4, 35.57, 6.38, 0, 48.04, -42.1], [9E9, 9E9, 9E9, 9E9, 9E9, 9E9]];
	VAR jointtarget SDP_1835 := [[7.59, 35.89, 5.85, 0, 48.26, -32.91], [9E9, 9E9, 9E9, 9E9, 9E9, 9E9]];
	VAR jointtarget SDP_1836 := [[7.73, 36.22, 5.27, 0, 48.5, -23.77], [9E9, 9E9, 9E9, 9E9, 9E9, 9E9]];
	VAR jointtarget SDP_1837 := [[7.82, 36.58, 4.65, 0, 48.76, -14.68], [9E9, 9E9, 9E9, 9E9, 9E9, 9E9]];
	VAR jointtarget SDP_1838 := [[7.85, 36.96, 4.01, 0, 49.03, -5.65], [9E9, 9E9, 9E9, 9E9, 9E9, 9E9]];
	VAR jointtarget SDP_1839 := [[7.83, 37.33, 3.37, 0, 49.3, 3.33], [9E9, 9E9, 9E9, 9E9, 9E9, 9E9]];
	VAR jointtarget SDP_1840 := [[7.68, 38.56, 1.24, 0, 50.2, 7.68], [9E9, 9E9, 9E9, 9E9, 9E9, 9E9]];
	VAR jointtarget SDP_1841 := [[7.54, 39.81, -0.94, 0, 51.13, 7.54], [9E9, 9E9, 9E9, 9E9, 9E9, 9E9]];
	VAR jointtarget SDP_1842 := [[7.4, 41.08, -3.16, 0, 52.08, 7.4], [9E9, 9E9, 9E9, 9E9, 9E9, 9E9]];
	VAR jointtarget SDP_1843 := [[7.27, 42.36, -5.43, 0, 53.06, 7.27], [9E9, 9E9, 9E9, 9E9, 9E9, 9E9]];
	VAR jointtarget SDP_1844 := [[7.15, 43.67, -7.75, 0, 54.07, 7.15], [9E9, 9E9, 9E9, 9E9, 9E9, 9E9]];
	VAR jointtarget SDP_1845 := [[7.02, 45.01, -10.13, 0, 55.12, 7.02], [9E9, 9E9, 9E9, 9E9, 9E9, 9E9]];
	VAR jointtarget SDP_1846 := [[6.9, 46.37, -12.57, 0, 56.2, 6.9], [9E9, 9E9, 9E9, 9E9, 9E9, 9E9]];
	VAR jointtarget SDP_1847 := [[6.79, 47.77, -15.08, 0, 57.31, 6.79], [9E9, 9E9, 9E9, 9E9, 9E9, 9E9]];
	VAR jointtarget SDP_1848 := [[6.68, 49.2, -17.67, 0, 58.47, 6.68], [9E9, 9E9, 9E9, 9E9, 9E9, 9E9]];
	VAR jointtarget SDP_1849 := [[6.57, 50.67, -20.35, 0, 59.67, 6.57], [9E9, 9E9, 9E9, 9E9, 9E9, 9E9]];
	VAR jointtarget SDP_1850 := [[6.56, 50.82, -20.61, 0, 59.79, 8.75], [9E9, 9E9, 9E9, 9E9, 9E9, 9E9]];
	VAR jointtarget SDP_1851 := [[6.54, 50.97, -20.88, 0, 59.91, 13.12], [9E9, 9E9, 9E9, 9E9, 9E9, 9E9]];
	VAR jointtarget SDP_1852 := [[6.51, 51.11, -21.14, 0, 60.03, 17.48], [9E9, 9E9, 9E9, 9E9, 9E9, 9E9]];
	VAR jointtarget SDP_1853 := [[6.48, 51.25, -21.4, 0, 60.15, 21.83], [9E9, 9E9, 9E9, 9E9, 9E9, 9E9]];
	VAR jointtarget SDP_1854 := [[6.44, 51.38, -21.64, 0, 60.26, 26.18], [9E9, 9E9, 9E9, 9E9, 9E9, 9E9]];
	VAR jointtarget SDP_1855 := [[6.39, 51.51, -21.88, 0, 60.37, 30.52], [9E9, 9E9, 9E9, 9E9, 9E9, 9E9]];
	VAR jointtarget SDP_1856 := [[6.34, 51.64, -22.11, 0, 60.47, 34.86], [9E9, 9E9, 9E9, 9E9, 9E9, 9E9]];
	VAR jointtarget SDP_1857 := [[6.28, 51.76, -22.32, 0, 60.57, 39.19], [9E9, 9E9, 9E9, 9E9, 9E9, 9E9]];
	VAR jointtarget SDP_1858 := [[6.22, 51.87, -22.52, 0, 60.66, 43.51], [9E9, 9E9, 9E9, 9E9, 9E9, 9E9]];
	VAR jointtarget SDP_1859 := [[6.15, 51.97, -22.71, 0, 60.74, 47.83], [9E9, 9E9, 9E9, 9E9, 9E9, 9E9]];
	VAR jointtarget SDP_1860 := [[6.11, 52.03, -22.82, 0, 60.79, 49.99], [9E9, 9E9, 9E9, 9E9, 9E9, 9E9]];
	VAR jointtarget SDP_1861 := [[6.07, 52.09, -22.93, 0, 60.84, 49.95], [9E9, 9E9, 9E9, 9E9, 9E9, 9E9]];
	VAR jointtarget SDP_1862 := [[6.03, 52.15, -23.04, 0, 60.89, 49.9], [9E9, 9E9, 9E9, 9E9, 9E9, 9E9]];
	VAR jointtarget SDP_1863 := [[5.99, 52.21, -23.15, 0, 60.94, 49.86], [9E9, 9E9, 9E9, 9E9, 9E9, 9E9]];
	VAR jointtarget SDP_1864 := [[5.94, 52.27, -23.26, 0, 60.99, 49.82], [9E9, 9E9, 9E9, 9E9, 9E9, 9E9]];
	VAR jointtarget SDP_1865 := [[5.9, 52.33, -23.37, 0, 61.04, 49.78], [9E9, 9E9, 9E9, 9E9, 9E9, 9E9]];
	VAR jointtarget SDP_1866 := [[5.86, 52.39, -23.48, 0, 61.09, 49.74], [9E9, 9E9, 9E9, 9E9, 9E9, 9E9]];
	VAR jointtarget SDP_1867 := [[5.82, 52.45, -23.59, 0, 61.14, 49.7], [9E9, 9E9, 9E9, 9E9, 9E9, 9E9]];
	VAR jointtarget SDP_1868 := [[5.78, 52.51, -23.7, 0, 61.19, 49.66], [9E9, 9E9, 9E9, 9E9, 9E9, 9E9]];
	VAR jointtarget SDP_1869 := [[5.74, 52.57, -23.81, 0, 61.24, 49.61], [9E9, 9E9, 9E9, 9E9, 9E9, 9E9]];
	VAR jointtarget SDP_1870 := [[5.58, 52.94, -24.49, 0, 61.55, 36.07], [9E9, 9E9, 9E9, 9E9, 9E9, 9E9]];
	VAR jointtarget SDP_1871 := [[5.54, 53.4, -25.32, 0, 61.93, 9.25], [9E9, 9E9, 9E9, 9E9, 9E9, 9E9]];
	VAR jointtarget SDP_1872 := [[5.62, 53.84, -26.14, 0, 62.3, -17.44], [9E9, 9E9, 9E9, 9E9, 9E9, 9E9]];
	VAR jointtarget SDP_1873 := [[5.8, 54.18, -26.76, 0, 62.58, -44.04], [9E9, 9E9, 9E9, 9E9, 9E9, 9E9]];
	VAR jointtarget SDP_1874 := [[6.04, 54.34, -27.05, 0, 62.71, -70.57], [9E9, 9E9, 9E9, 9E9, 9E9, 9E9]];
	VAR jointtarget SDP_1875 := [[6.3, 54.28, -26.94, 0, 62.66, -97.09], [9E9, 9E9, 9E9, 9E9, 9E9, 9E9]];
	VAR jointtarget SDP_1876 := [[6.51, 54.01, -26.46, 0, 62.44, -123.65], [9E9, 9E9, 9E9, 9E9, 9E9, 9E9]];
	VAR jointtarget SDP_1877 := [[6.64, 53.61, -25.71, 0, 62.1, -150.3], [9E9, 9E9, 9E9, 9E9, 9E9, 9E9]];
	VAR jointtarget SDP_1878 := [[6.66, 53.14, -24.86, 0, 61.72, -177.06], [9E9, 9E9, 9E9, 9E9, 9E9, 9E9]];
	VAR jointtarget SDP_1879 := [[6.55, 52.72, -24.09, 0, 61.37, -203.94], [9E9, 9E9, 9E9, 9E9, 9E9, 9E9]];
	VAR jointtarget SDP_1880 := [[6.52, 52.65, -23.95, 0, 61.3, -217.36], [9E9, 9E9, 9E9, 9E9, 9E9, 9E9]];
	VAR jointtarget SDP_1881 := [[6.48, 52.57, -23.82, 0, 61.24, -217.39], [9E9, 9E9, 9E9, 9E9, 9E9, 9E9]];
	VAR jointtarget SDP_1882 := [[6.45, 52.5, -23.68, 0, 61.18, -217.42], [9E9, 9E9, 9E9, 9E9, 9E9, 9E9]];
	VAR jointtarget SDP_1883 := [[6.42, 52.43, -23.54, 0, 61.12, -217.46], [9E9, 9E9, 9E9, 9E9, 9E9, 9E9]];
	VAR jointtarget SDP_1884 := [[6.39, 52.35, -23.41, 0, 61.06, -217.49], [9E9, 9E9, 9E9, 9E9, 9E9, 9E9]];
	VAR jointtarget SDP_1885 := [[6.35, 52.28, -23.27, 0, 61, -217.52], [9E9, 9E9, 9E9, 9E9, 9E9, 9E9]];
	VAR jointtarget SDP_1886 := [[6.32, 52.2, -23.14, 0, 60.93, -217.56], [9E9, 9E9, 9E9, 9E9, 9E9, 9E9]];
	VAR jointtarget SDP_1887 := [[6.29, 52.13, -23, 0, 60.87, -217.59], [9E9, 9E9, 9E9, 9E9, 9E9, 9E9]];
	VAR jointtarget SDP_1888 := [[6.25, 52.06, -22.87, 0, 60.81, -217.62], [9E9, 9E9, 9E9, 9E9, 9E9, 9E9]];
	VAR jointtarget SDP_1889 := [[6.22, 51.98, -22.74, 0, 60.75, -217.66], [9E9, 9E9, 9E9, 9E9, 9E9, 9E9]];
	VAR jointtarget SDP_1890 := [[6.17, 51.86, -22.51, 0, 60.65, -215.51], [9E9, 9E9, 9E9, 9E9, 9E9, 9E9]];
	VAR jointtarget SDP_1891 := [[6.12, 51.73, -22.27, 0, 60.54, -211.17], [9E9, 9E9, 9E9, 9E9, 9E9, 9E9]];
	VAR jointtarget SDP_1892 := [[6.08, 51.59, -22.02, 0, 60.43, -206.83], [9E9, 9E9, 9E9, 9E9, 9E9, 9E9]];
	VAR jointtarget SDP_1893 := [[6.05, 51.45, -21.77, 0, 60.31, -202.47], [9E9, 9E9, 9E9, 9E9, 9E9, 9E9]];
	VAR jointtarget SDP_1894 := [[6.02, 51.31, -21.5, 0, 60.2, -198.11], [9E9, 9E9, 9E9, 9E9, 9E9, 9E9]];
	VAR jointtarget SDP_1895 := [[6, 51.16, -21.24, 0, 60.07, -193.75], [9E9, 9E9, 9E9, 9E9, 9E9, 9E9]];
	VAR jointtarget SDP_1896 := [[5.98, 51.01, -20.97, 0, 59.95, -189.38], [9E9, 9E9, 9E9, 9E9, 9E9, 9E9]];
	VAR jointtarget SDP_1897 := [[5.97, 50.86, -20.7, 0, 59.83, -185], [9E9, 9E9, 9E9, 9E9, 9E9, 9E9]];
	VAR jointtarget SDP_1898 := [[5.97, 50.72, -20.42, 0, 59.71, -180.61], [9E9, 9E9, 9E9, 9E9, 9E9, 9E9]];
	VAR jointtarget SDP_1899 := [[5.98, 50.57, -20.15, 0, 59.59, -176.22], [9E9, 9E9, 9E9, 9E9, 9E9, 9E9]];
	VAR jointtarget SDP_1900 := [[6.07, 49.19, -17.65, 0, 58.46, -173.93], [9E9, 9E9, 9E9, 9E9, 9E9, 9E9]];
	VAR jointtarget SDP_1901 := [[6.16, 47.85, -15.22, 0, 57.38, -173.84], [9E9, 9E9, 9E9, 9E9, 9E9, 9E9]];
	VAR jointtarget SDP_1902 := [[6.26, 46.54, -12.86, 0, 56.33, -173.74], [9E9, 9E9, 9E9, 9E9, 9E9, 9E9]];
	VAR jointtarget SDP_1903 := [[6.36, 45.25, -10.57, 0, 55.31, -173.64], [9E9, 9E9, 9E9, 9E9, 9E9, 9E9]];
	VAR jointtarget SDP_1904 := [[6.47, 44, -8.33, 0, 54.33, -173.53], [9E9, 9E9, 9E9, 9E9, 9E9, 9E9]];
	VAR jointtarget SDP_1905 := [[6.57, 42.77, -6.14, 0, 53.37, -173.43], [9E9, 9E9, 9E9, 9E9, 9E9, 9E9]];
	VAR jointtarget SDP_1906 := [[6.68, 41.55, -4, 0, 52.44, -173.32], [9E9, 9E9, 9E9, 9E9, 9E9, 9E9]];
	VAR jointtarget SDP_1907 := [[6.8, 40.36, -1.9, 0, 51.54, -173.2], [9E9, 9E9, 9E9, 9E9, 9E9, 9E9]];
	VAR jointtarget SDP_1908 := [[6.92, 39.18, 0.16, 0, 50.66, -173.08], [9E9, 9E9, 9E9, 9E9, 9E9, 9E9]];
	VAR jointtarget SDP_1909 := [[7.04, 38.02, 2.17, 0, 49.8, -172.96], [9E9, 9E9, 9E9, 9E9, 9E9, 9E9]];
	VAR jointtarget SDP_1910 := [[7.05, 37.64, 2.83, 0, 49.53, -177.45], [9E9, 9E9, 9E9, 9E9, 9E9, 9E9]];
	VAR jointtarget SDP_1911 := [[7.02, 37.27, 3.47, 0, 49.26, -186.48], [9E9, 9E9, 9E9, 9E9, 9E9, 9E9]];
	VAR jointtarget SDP_1912 := [[6.93, 36.91, 4.09, 0, 49, -195.57], [9E9, 9E9, 9E9, 9E9, 9E9, 9E9]];
	VAR jointtarget SDP_1913 := [[6.78, 36.57, 4.68, 0, 48.75, -204.72], [9E9, 9E9, 9E9, 9E9, 9E9, 9E9]];
	VAR jointtarget SDP_1914 := [[6.6, 36.26, 5.21, 0, 48.53, -213.9], [9E9, 9E9, 9E9, 9E9, 9E9, 9E9]];
	VAR jointtarget SDP_1915 := [[6.36, 35.99, 5.68, 0, 48.34, -223.14], [9E9, 9E9, 9E9, 9E9, 9E9, 9E9]];
	VAR jointtarget SDP_1916 := [[6.09, 35.76, 6.06, 0, 48.17, -232.41], [9E9, 9E9, 9E9, 9E9, 9E9, 9E9]];
	VAR jointtarget SDP_1917 := [[5.79, 35.59, 6.36, 0, 48.05, -241.71], [9E9, 9E9, 9E9, 9E9, 9E9, 9E9]];
	VAR jointtarget SDP_1918 := [[5.47, 35.46, 6.57, 0, 47.96, -251.03], [9E9, 9E9, 9E9, 9E9, 9E9, 9E9]];
	VAR jointtarget SDP_1919 := [[5.13, 35.4, 6.68, 0, 47.92, -260.37], [9E9, 9E9, 9E9, 9E9, 9E9, 9E9]];
	VAR jointtarget SDP_1920 := [[4.05, 35.31, 6.84, 0, 47.85, -265.95], [9E9, 9E9, 9E9, 9E9, 9E9, 9E9]];
	VAR jointtarget SDP_1921 := [[2.97, 35.24, 6.96, 0, 47.8, -267.03], [9E9, 9E9, 9E9, 9E9, 9E9, 9E9]];
	VAR jointtarget SDP_1922 := [[1.89, 35.19, 7.04, 0, 47.77, -268.11], [9E9, 9E9, 9E9, 9E9, 9E9, 9E9]];
	VAR jointtarget SDP_1923 := [[0.8, 35.16, 7.09, 0, 47.75, -269.2], [9E9, 9E9, 9E9, 9E9, 9E9, 9E9]];
	VAR jointtarget SDP_1924 := [[-0.28, 35.16, 7.1, 0, 47.75, -270.28], [9E9, 9E9, 9E9, 9E9, 9E9, 9E9]];
	VAR jointtarget SDP_1925 := [[-1.37, 35.17, 7.07, 0, 47.76, -271.37], [9E9, 9E9, 9E9, 9E9, 9E9, 9E9]];
	VAR jointtarget SDP_1926 := [[-2.45, 35.21, 7, 0, 47.79, -272.45], [9E9, 9E9, 9E9, 9E9, 9E9, 9E9]];
	VAR jointtarget SDP_1927 := [[-3.53, 35.27, 6.9, 0, 47.83, -273.53], [9E9, 9E9, 9E9, 9E9, 9E9, 9E9]];
	VAR jointtarget SDP_1928 := [[-4.61, 35.35, 6.76, 0, 47.89, -274.61], [9E9, 9E9, 9E9, 9E9, 9E9, 9E9]];
	VAR jointtarget SDP_1929 := [[-5.69, 35.46, 6.58, 0, 47.96, -275.69], [9E9, 9E9, 9E9, 9E9, 9E9, 9E9]];
	VAR jointtarget SDP_1930 := [[-5.72, 35.46, 6.58, 0, 47.96, -276.38], [9E9, 9E9, 9E9, 9E9, 9E9, 9E9]];
	VAR jointtarget SDP_1931 := [[-5.75, 35.47, 6.57, 0, 47.97, -277.74], [9E9, 9E9, 9E9, 9E9, 9E9, 9E9]];
	VAR jointtarget SDP_1932 := [[-5.79, 35.47, 6.56, 0, 47.97, -279.1], [9E9, 9E9, 9E9, 9E9, 9E9, 9E9]];
	VAR jointtarget SDP_1933 := [[-5.82, 35.48, 6.55, 0, 47.97, -280.46], [9E9, 9E9, 9E9, 9E9, 9E9, 9E9]];
	VAR jointtarget SDP_1934 := [[-5.85, 35.49, 6.53, 0, 47.98, -281.81], [9E9, 9E9, 9E9, 9E9, 9E9, 9E9]];
	VAR jointtarget SDP_1935 := [[-5.89, 35.5, 6.52, 0, 47.99, -283.17], [9E9, 9E9, 9E9, 9E9, 9E9, 9E9]];
	VAR jointtarget SDP_1936 := [[-5.92, 35.5, 6.5, 0, 47.99, -284.53], [9E9, 9E9, 9E9, 9E9, 9E9, 9E9]];
	VAR jointtarget SDP_1937 := [[-5.95, 35.51, 6.49, 0, 48, -285.88], [9E9, 9E9, 9E9, 9E9, 9E9, 9E9]];
	VAR jointtarget SDP_1938 := [[-5.98, 35.53, 6.47, 0, 48.01, -287.24], [9E9, 9E9, 9E9, 9E9, 9E9, 9E9]];
	VAR jointtarget SDP_1939 := [[-6.02, 35.54, 6.45, 0, 48.01, -288.59], [9E9, 9E9, 9E9, 9E9, 9E9, 9E9]];
	VAR jointtarget SDP_1940 := [[-6.14, 35.59, 6.37, 0, 48.05, -289.38], [9E9, 9E9, 9E9, 9E9, 9E9, 9E9]];
	VAR jointtarget SDP_1941 := [[-6.27, 35.63, 6.28, 0, 48.08, -289.51], [9E9, 9E9, 9E9, 9E9, 9E9, 9E9]];
	VAR jointtarget SDP_1942 := [[-6.4, 35.68, 6.2, 0, 48.12, -289.64], [9E9, 9E9, 9E9, 9E9, 9E9, 9E9]];
	VAR jointtarget SDP_1943 := [[-6.53, 35.73, 6.11, 0, 48.15, -289.77], [9E9, 9E9, 9E9, 9E9, 9E9, 9E9]];
	VAR jointtarget SDP_1944 := [[-6.66, 35.78, 6.03, 0, 48.19, -289.9], [9E9, 9E9, 9E9, 9E9, 9E9, 9E9]];
	VAR jointtarget SDP_1945 := [[-6.78, 35.83, 5.94, 0, 48.22, -290.02], [9E9, 9E9, 9E9, 9E9, 9E9, 9E9]];
	VAR jointtarget SDP_1946 := [[-6.91, 35.88, 5.86, 0, 48.26, -290.15], [9E9, 9E9, 9E9, 9E9, 9E9, 9E9]];
	VAR jointtarget SDP_1947 := [[-7.04, 35.93, 5.77, 0, 48.3, -290.28], [9E9, 9E9, 9E9, 9E9, 9E9, 9E9]];
	VAR jointtarget SDP_1948 := [[-7.16, 35.98, 5.68, 0, 48.33, -290.4], [9E9, 9E9, 9E9, 9E9, 9E9, 9E9]];
	VAR jointtarget SDP_1949 := [[-7.29, 36.04, 5.59, 0, 48.37, -290.53], [9E9, 9E9, 9E9, 9E9, 9E9, 9E9]];
	VAR jointtarget SDP_1950 := [[-7.55, 36.09, 5.51, 0, 48.41, -280.46], [9E9, 9E9, 9E9, 9E9, 9E9, 9E9]];
	VAR jointtarget SDP_1951 := [[-7.8, 36.04, 5.59, 0, 48.37, -260.07], [9E9, 9E9, 9E9, 9E9, 9E9, 9E9]];
	VAR jointtarget SDP_1952 := [[-8.03, 35.89, 5.84, 0, 48.27, -239.65], [9E9, 9E9, 9E9, 9E9, 9E9, 9E9]];
	VAR jointtarget SDP_1953 := [[-8.2, 35.67, 6.22, 0, 48.11, -219.17], [9E9, 9E9, 9E9, 9E9, 9E9, 9E9]];
	VAR jointtarget SDP_1954 := [[-8.28, 35.4, 6.68, 0, 47.92, -198.6], [9E9, 9E9, 9E9, 9E9, 9E9, 9E9]];
	VAR jointtarget SDP_1955 := [[-8.27, 35.12, 7.16, 0, 47.72, -177.95], [9E9, 9E9, 9E9, 9E9, 9E9, 9E9]];
	VAR jointtarget SDP_1956 := [[-8.17, 34.86, 7.6, 0, 47.54, -157.19], [9E9, 9E9, 9E9, 9E9, 9E9, 9E9]];
	VAR jointtarget SDP_1957 := [[-7.98, 34.66, 7.95, 0, 47.4, -136.36], [9E9, 9E9, 9E9, 9E9, 9E9, 9E9]];
	VAR jointtarget SDP_1958 := [[-7.74, 34.54, 8.15, 0, 47.31, -115.47], [9E9, 9E9, 9E9, 9E9, 9E9, 9E9]];
	VAR jointtarget SDP_1959 := [[-7.47, 34.51, 8.19, 0, 47.29, -94.56], [9E9, 9E9, 9E9, 9E9, 9E9, 9E9]];
